KUKA KRL program: Glode_HanGao.src, Glode_HanGao.dat

--- Glode_HanGao.src ---
&ACCESS RVO1
&REL 506
&PARAM EDITMASK = *
&PARAM TEMPLATE = C:\KRC\Roboter\Template\vorgabe
&PARAM DISKPATH = KRC:\R1\Program\HG
DEF Glode_HanGao( )

;# DATE:2021-1-4


END



GLOBAL DEF Vision_Path(PATH_POS:OUT,POS_OFFSET:IN)
DECL E6POS PATH_POS,POS_OFFSET

;Halt


IF Vision_OFFSET_STATE==FALSE THEN
 PATH_POS=POS_OFFSET:PATH_POS
ENDIF

Vision_OFFSET_STATE=TRUE



END
GLOBAL DEF Vision_EndPath(PATH_POS:OUT,POS_OFFSET:IN)
DECL E6POS PATH_POS,POS_OFFSET

;HALT
INTERRUPT OFF 20
PATH_POS=INV_Pos(POS_OFFSET):PATH_POS



END



GLOBAL DEF Vision_Results_Pos(Vision_PATH:IN,Result_Pos:IN,POS_Offset:OUT)
DECL E6POS POS_Offset,Result_Pos,Offset,Error_Offset,Result_Pos_Inv
DECL Vision_PATH_Enum Vision_PATH
DECL INT Result_ID,OPFFSET
DECL CHAR POS_Sting[1024],Message_Show[1024]
DECL State_t _State
DECL VAR_STATE VarT

Message_Show[]=" "
OPFFSET=0
Offset=$NULLFRAME
Error_Offset=$NULLFRAME

IF Vision_Type ==#Vision_Run THEN


VarT=VARSTATE("POS_Offset")
SWITCH VarT

CASE #DECLARED

RETURN

CASE #INITIALIZED

;Result_Pos_Inv=Inv_Pos(Result_Pos)

Error_Offset=Inv_Pos(Result_Pos):Pos_Offset
;Halt

;Offset.X=Error_Offset.X-POS_Offset.X
;Offset.Y=Error_Offset.Y-POS_Offset.Y
;Offset.Z=Error_Offset.z-POS_Offset.Z
;Offset.A=Error_Offset.A-POS_Offset.A
;Offset.B=Error_Offset.B-POS_Offset.B
;Offset.C=Error_Offset.C-POS_Offset.C





SWITCH Vision_PATH
CASE #X

SWRITE( Message_Show[] , _State , OPFFSET ,"Vision Find  Offset: X:%7.3F Translation Max:%7.3F," ,Error_Offset.X, Vision_Trans_Max_Offset  )

if (ABS(Error_Offset.X)<Vision_Trans_Max_Offset)  THEN

POS_Offset.X=Result_Pos.X
ELSE


MsgQuit(Message_Show[], "HanGao")
RETURN
ENDIF


CASE #Y

SWRITE( Message_Show[] , _State , OPFFSET ,"Vision Find  Offset: Y:%7.3F Translation Max:%7.3F," ,Error_Offset.Y, Vision_Trans_Max_Offset  )
if (ABS(Error_Offset.Y)<Vision_Trans_Max_Offset)  THEN

POS_Offset.Y=Result_Pos.Y
ELSE


MsgQuit(Message_Show[], "HanGao")
RETURN
ENDIF
CASE #Z
SWRITE( Message_Show[] , _State , OPFFSET ,"Vision Find  Offset: Z:%7.3F Translation Max:%7.3F," ,Error_Offset.Z, Vision_Trans_Max_Offset  )
if (ABS(Error_Offset.Z)<Vision_Trans_Max_Offset)  THEN

POS_Offset.Z=Result_Pos.Z
ELSE


MsgQuit(Message_Show[], "HanGao")
RETURN
ENDIF
CASE #XY

SWRITE( Message_Show[] , _State , OPFFSET ,"Vision Find  Offset: X:%7.3F,Y:%7.3F Translation Max:%7.3F" ,Error_Offset.X,Error_Offset.Y ,Vision_Trans_Max_Offset  )

if (ABS(Error_Offset.X)<Vision_Trans_Max_Offset) AND (ABS(Error_Offset.Y)<Vision_Trans_Max_Offset)  THEN

POS_Offset.X=Result_Pos.X
POS_Offset.Y=Result_Pos.Y
ELSE


MsgQuit(Message_Show[], "HanGao")
RETURN
ENDIF
CASE #XZ

SWRITE( Message_Show[] , _State , OPFFSET ,"Vision Find  Offset: X:%7.3F,Z:%7.3F Translation Max:%7.3F" ,Error_Offset.X,Error_Offset.Z, Vision_Trans_Max_Offset  )

if (ABS(Error_Offset.X)<Vision_Trans_Max_Offset) AND (ABS(Error_Offset.Z)<Vision_Trans_Max_Offset)  THEN

POS_Offset.X=Result_Pos.X
POS_Offset.Z=Result_Pos.Z
ELSE


MsgQuit(Message_Show[], "HanGao")
RETURN
ENDIF
CASE #YZ

SWRITE( Message_Show[] , _State , OPFFSET ,"Vision Find  Offset: Y:%7.3F,Z:%7.3F Translation Max:%7.3F" ,Error_Offset.Y,Error_Offset.Z, Vision_Trans_Max_Offset  )

if (ABS(Error_Offset.Y)<Vision_Trans_Max_Offset) AND (ABS(Error_Offset.Y)<Vision_Trans_Max_Offset)  THEN

POS_Offset.Y=Result_Pos.Y
POS_Offset.Z=Result_Pos.Z
ELSE


MsgQuit(Message_Show[], "HanGao")
RETURN
ENDIF
CASE #XYZ

SWRITE( Message_Show[] , _State , OPFFSET ,"Vision Find  Offset: X:%7.3F,Y:%7.3F,Z:%7.3F Translation Max:%7.3F" ,Error_Offset.X,Error_Offset.Y,Error_Offset.Z, Vision_Trans_Max_Offset  )

if (ABS(Error_Offset.X)<Vision_Trans_Max_Offset) AND (ABS(Error_Offset.Y)<Vision_Trans_Max_Offset) AND (ABS(Error_Offset.Z)<Vision_Trans_Max_Offset)   THEN

POS_Offset.X=Result_Pos.X
POS_Offset.Y=Result_Pos.Y
POS_Offset.Z=Result_Pos.Z
ELSE


MsgQuit(Message_Show[], "HanGao")
RETURN
ENDIF
CASE #XYZABC

SWRITE( Message_Show[] , _State , OPFFSET ,"Vision Find  Offset: X:%7.3F,Y:%7.3F,Z:%7.3F,A:%7.3F,B:%7.3F,C:%7.3F Translation Max:%7.3F,Rotation Max:%7.3F" ,Error_Offset.X,Error_Offset.Y,Error_Offset.Z,Error_Offset.A,Error_Offset.B,Error_Offset.C, Vision_Trans_Max_Offset ,Vision_Rota_Max_Offset )


if (ABS(Error_Offset.X)<Vision_Trans_Max_Offset) AND (ABS(Error_Offset.Y)<Vision_Trans_Max_Offset) AND (ABS(Error_Offset.Z)<Vision_Trans_Max_Offset) AND (ABS(Error_Offset.A)<Vision_Rota_Max_Offset) AND (ABS(Error_Offset.B)<Vision_Rota_Max_Offset) AND (ABS(Error_Offset.C)<Vision_Rota_Max_Offset)  THEN

POS_Offset.X=Result_Pos.X
POS_Offset.Y=Result_Pos.Y
POS_Offset.Z=Result_Pos.Z
POS_Offset.A=Result_Pos.A
POS_Offset.B=Result_Pos.B
POS_Offset.C=Result_Pos.C

ELSE

MsgQuit(Message_Show[], "HanGao")
RETURN
ENDIF
ENDSWITCH



MSGNOTIFY(Message_Show[])



CASE #UNKNOWN

RETURN

ENDSWITCH


ENDIF



;ENDIF

END
GLOBAL DEF Vision_Results_Offset(Vision_PATH:IN,POS_Offset_1:OUT,POS_Offset_2:OUT,POS_Offset_3:OUT,POS_Offset_4:OUT,POS_Offset_5:OUT,POS_Offset_6:OUT,POS_Offset_7:OUT,POS_Offset_8:OUT,POS_Offset_9:OUT)
DECL E6POS POS_Offset_1 ,POS_Offset_2,POS_Offset_3,POS_Offset_4,POS_Offset_5,POS_Offset_6,POS_Offset_7,POS_Offset_8,POS_Offset_9
DECL Vision_PATH_Enum Vision_PATH
DECL INT Result_ID

IF Vision_Type ==#Vision_Run THEN



Vision_Results_Pos(Vision_PATH,Vision_Result_POS,POS_Offset_1)
Vision_Results_Pos(Vision_PATH,Vision_Result_POS,POS_Offset_2)
Vision_Results_Pos(Vision_PATH,Vision_Result_POS,POS_Offset_3)
Vision_Results_Pos(Vision_PATH,Vision_Result_POS,POS_Offset_4)
Vision_Results_Pos(Vision_PATH,Vision_Result_POS,POS_Offset_5)
Vision_Results_Pos(Vision_PATH,Vision_Result_POS,POS_Offset_6)
Vision_Results_Pos(Vision_PATH,Vision_Result_POS,POS_Offset_7)
Vision_Results_Pos(Vision_PATH,Vision_Result_POS,POS_Offset_8)
Vision_Results_Pos(Vision_PATH,Vision_Result_POS,POS_Offset_9)
ENDIF




END






GLOBAL DEF HanGao_Surr_Calculate(Surr_Path:IN , Sink_Area:IN ,POS_Type:IN , Lin_Pos:OUt , Cir_Middle_POS:OUT , Cir_END_POS:OUT , Offset_info:OUT  ,Offset_cir_info:out , Offset_No:IN , Work_Area:IN, Sink_Type:IN)
;------------DECL_VALUE--------------
DECL REAL Surr_Path
DECL Sink_Type_Enum  Sink_Type
DECL Area_Enum Sink_Area
DECL E6POS Lin_Pos
DECL E6POS Cir_Middle_POS
DECL E6POS Cir_END_POS
DECL Pos_Type_Enum Pos_Type
DECL Offset_POS Offset_info , Offset_cir_info
DECL Surround_Welding_Type Sink_Welding_Size
DECL INT OFFSET_NO,Work_Area

;------------DECL_VALUE--------------





Lin_Pos={X 0,Y 0, Z 0,A 0,B 0,C 0}

Cir_Middle_POS={X 0,Y 0, Z 0,A 0,B 0,C 0}

Cir_END_POS={X 0,Y 0, Z 0,A 0,B 0,C 0}


switch Work_Area

CASE 1
Sink_Welding_Size=N1_Sink_Data

CASE 2
Sink_Welding_Size=N2_Sink_Data

ENDSWITCH



SWITCH Sink_Area

CASE #L0





 UL_Equation(N315_OFFSET_POS,N45_OFFSET_POS,(Surr_Path*0.01),Sink_Welding_Size.Sink_Size_R,Lin_Pos)



 ;Lin_Pos.X=Sink_Welding_Size.Sink_Size_Width+Sink_Welding_Size.Sink_Size_Down_Distance
 ;Lin_Pos.Y=(Sink_Welding_Size.Sink_Size_Long-Sink_Welding_Size.Sink_Size_R*2)* (1-(Surr_Path*0.01))+Sink_Welding_Size.Sink_Size_Left_Distance+Sink_Welding_Size.Sink_Size_R
 Lin_Pos.Z=-(Sink_Welding_Size.Sink_Size_Panel_Thick)

 Lin_Pos.A=0
 Lin_Pos.B=L0_Welding_Craft[Work_Area,OFFSET_NO].Welding_Angle
 Lin_Pos.C=0


L0_Welding_Craft[Work_Area,OFFSET_NO].Welding_Pos.X=Lin_Pos.X
L0_Welding_Craft[Work_Area,OFFSET_NO].Welding_Pos.Y=Lin_Pos.Y
L0_Welding_Craft[Work_Area,OFFSET_NO].Welding_Pos.Z=Lin_Pos.Z
L0_Welding_Craft[Work_Area,OFFSET_NO].Welding_Pos.A=Lin_Pos.A
L0_Welding_Craft[Work_Area,OFFSET_NO].Welding_Pos.B=Lin_Pos.B
L0_Welding_Craft[Work_Area,OFFSET_NO].Welding_Pos.C=Lin_Pos.C
CASE #C45


SWITCH Pos_Type

CASE #C_LIN_POS


UL_Equation(N315_OFFSET_POS,N45_OFFSET_POS,1,Sink_Welding_Size.Sink_Size_R,Lin_Pos)

;Lin_Pos.X=Sink_Welding_Size.Sink_Size_Width+Sink_Welding_Size.Sink_Size_Down_Distance
;Lin_Pos.Y=Sink_Welding_Size.Sink_Size_Left_Distance+Sink_Welding_Size.Sink_Size_R
Lin_Pos.Z=-(Sink_Welding_Size.Sink_Size_Panel_Thick)

Lin_Pos.A=0
Lin_Pos.B=C45_Welding_Craft[Work_Area,1].Welding_Angle
Lin_Pos.C=0

C45_Welding_Craft[Work_Area,1].Welding_Pos.X=Lin_Pos.X
C45_Welding_Craft[Work_Area,1].Welding_Pos.Y=Lin_Pos.Y
C45_Welding_Craft[Work_Area,1].Welding_Pos.Z=Lin_Pos.Z
C45_Welding_Craft[Work_Area,1].Welding_Pos.A=Lin_Pos.A
C45_Welding_Craft[Work_Area,1].Welding_Pos.B=Lin_Pos.B
C45_Welding_Craft[Work_Area,1].Welding_Pos.C=Lin_Pos.C

CASE #C_CIR_POS


 Cir_Middle_POS.X=N45_CIR_POS.x
 Cir_Middle_POS.Y=N45_CIR_POS.Y

 ;Cir_Middle_POS.x=Sink_Welding_Size.Sink_Size_Down_Distance+Sink_Welding_Size.Sink_Size_Width-Sink_Welding_Size.Sink_Size_R+(COS(45)*Sink_Welding_Size.Sink_Size_R)
 ;Cir_Middle_POS.Y=Sink_Welding_Size.Sink_Size_Left_Distance+((1-COS(45))*Sink_Welding_Size.Sink_Size_R)
 Cir_Middle_POS.Z=-(Sink_Welding_Size.Sink_Size_Panel_Thick)


 UL_Equation(N45_OFFSET_POS,N135_OFFSET_POS,0,Sink_Welding_Size.Sink_Size_R,Cir_END_POS)

 ;Cir_END_POS.X=Sink_Welding_Size.Sink_Size_Down_Distance+Sink_Welding_Size.Sink_Size_Width-Sink_Welding_Size.Sink_Size_R
 ;Cir_END_POS.Y=Sink_Welding_Size.Sink_Size_Left_Distance
 Cir_END_POS.Z=-(Sink_Welding_Size.Sink_Size_Panel_Thick)


 Cir_END_POS.A=0
 Cir_END_POS.B=0
 Cir_END_POS.C=C45_Welding_Craft[Work_Area,3].Welding_Angle



C45_Welding_Craft[Work_Area,2].Welding_Pos.X=Cir_Middle_POS.X
C45_Welding_Craft[Work_Area,2].Welding_Pos.Y=Cir_Middle_POS.Y
C45_Welding_Craft[Work_Area,2].Welding_Pos.Z=Cir_Middle_POS.Z
C45_Welding_Craft[Work_Area,2].Welding_Pos.A=Cir_Middle_POS.A
C45_Welding_Craft[Work_Area,2].Welding_Pos.B=Cir_Middle_POS.B
C45_Welding_Craft[Work_Area,2].Welding_Pos.C=Cir_Middle_POS.C

C45_Welding_Craft[Work_Area,3].Welding_Pos.X=Cir_END_POS.X
C45_Welding_Craft[Work_Area,3].Welding_Pos.Y=Cir_END_POS.Y
C45_Welding_Craft[Work_Area,3].Welding_Pos.Z=Cir_END_POS.Z
C45_Welding_Craft[Work_Area,3].Welding_Pos.A=Cir_END_POS.A
C45_Welding_Craft[Work_Area,3].Welding_Pos.B=Cir_END_POS.B
C45_Welding_Craft[Work_Area,3].Welding_Pos.C=Cir_END_POS.C

ENDSWITCH


CASE #L90


UL_Equation(N45_OFFSET_POS,N135_OFFSET_POS,(Surr_Path*0.01),Sink_Welding_Size.Sink_Size_R, Lin_Pos)

 ;Lin_Pos.X=(Sink_Welding_Size.Sink_Size_Width-Sink_Welding_Size.Sink_Size_R*2)* (1-(Surr_Path*0.01))+Sink_Welding_Size.Sink_Size_Down_Distance+Sink_Welding_Size.Sink_Size_R
 ;Lin_Pos.Y=Sink_Welding_Size.Sink_Size_Left_Distance
 Lin_Pos.Z=-(Sink_Welding_Size.Sink_Size_Panel_Thick)
 Lin_Pos.A=0
 Lin_Pos.B=0
 Lin_Pos.C=L90_Welding_Craft[Work_Area,OFFSET_NO].Welding_Angle

L90_Welding_Craft[Work_Area,OFFSET_NO].Welding_Pos.X=Lin_Pos.X
L90_Welding_Craft[Work_Area,OFFSET_NO].Welding_Pos.Y=Lin_Pos.Y
L90_Welding_Craft[Work_Area,OFFSET_NO].Welding_Pos.Z=Lin_Pos.Z
L90_Welding_Craft[Work_Area,OFFSET_NO].Welding_Pos.A=Lin_Pos.A
L90_Welding_Craft[Work_Area,OFFSET_NO].Welding_Pos.B=Lin_Pos.B
L90_Welding_Craft[Work_Area,OFFSET_NO].Welding_Pos.C=Lin_Pos.C

CASE #C135

SWITCH Pos_Type

CASE #C_LIN_POS

UL_Equation(N45_OFFSET_POS,N135_OFFSET_POS,1,Sink_Welding_Size.Sink_Size_R, Lin_Pos)

 ;Lin_Pos.X=Sink_Welding_Size.Sink_Size_Down_Distance+Sink_Welding_Size.Sink_Size_R
 ;Lin_Pos.Y=Sink_Welding_Size.Sink_Size_Left_Distance
 Lin_Pos.Z=-(Sink_Welding_Size.Sink_Size_Panel_Thick)
 Lin_Pos.A=0
 Lin_Pos.B=0
 Lin_Pos.C=C135_Welding_Craft[Work_Area,1].Welding_Angle

C135_Welding_Craft[Work_Area,1].Welding_Pos.X=Lin_Pos.X
C135_Welding_Craft[Work_Area,1].Welding_Pos.Y=Lin_Pos.Y
C135_Welding_Craft[Work_Area,1].Welding_Pos.Z=Lin_Pos.Z
C135_Welding_Craft[Work_Area,1].Welding_Pos.A=Lin_Pos.A
C135_Welding_Craft[Work_Area,1].Welding_Pos.B=Lin_Pos.B
C135_Welding_Craft[Work_Area,1].Welding_Pos.C=Lin_Pos.C

CASE #C_CIR_POS



 Cir_Middle_POS.X=N135_CIR_POS.x
 Cir_Middle_POS.Y=N135_CIR_POS.Y


 ;Cir_Middle_POS.x=Sink_Welding_Size.Sink_Size_Down_Distance+((1-COS(45))*Sink_Welding_Size.Sink_Size_R)
 ;Cir_Middle_POS.Y=Sink_Welding_Size.Sink_Size_Left_Distance+((1-COS(45))*Sink_Welding_Size.Sink_Size_R)
 Cir_Middle_POS.Z=-(Sink_Welding_Size.Sink_Size_Panel_Thick)



 UL_Equation(N135_OFFSET_POS,N225_OFFSET_POS,0,Sink_Welding_Size.Sink_Size_R,Cir_END_POS)

 ;Cir_END_POS.X=Sink_Welding_Size.Sink_Size_Down_Distance
 ;Cir_END_POS.Y=Sink_Welding_Size.Sink_Size_Left_Distance+Sink_Welding_Size.Sink_Size_R
 Cir_END_POS.Z=-(Sink_Welding_Size.Sink_Size_Panel_Thick)
 Cir_END_POS.A=0
 Cir_END_POS.B=C135_Welding_Craft[Work_Area,3].Welding_Angle
 Cir_END_POS.C=0

C135_Welding_Craft[Work_Area,2].Welding_Pos.X=Cir_Middle_POS.X
C135_Welding_Craft[Work_Area,2].Welding_Pos.Y=Cir_Middle_POS.Y
C135_Welding_Craft[Work_Area,2].Welding_Pos.Z=Cir_Middle_POS.Z
C135_Welding_Craft[Work_Area,2].Welding_Pos.A=Cir_Middle_POS.A
C135_Welding_Craft[Work_Area,2].Welding_Pos.B=Cir_Middle_POS.B
C135_Welding_Craft[Work_Area,2].Welding_Pos.C=Cir_Middle_POS.C

C135_Welding_Craft[Work_Area,3].Welding_Pos.X=Cir_END_POS.X
C135_Welding_Craft[Work_Area,3].Welding_Pos.Y=Cir_END_POS.Y
C135_Welding_Craft[Work_Area,3].Welding_Pos.Z=Cir_END_POS.Z
C135_Welding_Craft[Work_Area,3].Welding_Pos.A=Cir_END_POS.A
C135_Welding_Craft[Work_Area,3].Welding_Pos.B=Cir_END_POS.B
C135_Welding_Craft[Work_Area,3].Welding_Pos.C=Cir_END_POS.C

ENDSWITCH


CASE #L180

UL_Equation(N135_OFFSET_POS,N225_OFFSET_POS,(Surr_Path*0.01),Sink_Welding_Size.Sink_Size_R, Lin_Pos)

 ;Lin_Pos.X=Sink_Welding_Size.Sink_Size_Down_Distance
 ;Lin_Pos.Y=(Sink_Welding_Size.Sink_Size_Long-Sink_Welding_Size.Sink_Size_R*2)* (Surr_Path*0.01)+Sink_Welding_Size.Sink_Size_Left_Distance+Sink_Welding_Size.Sink_Size_R
 Lin_Pos.Z=-(Sink_Welding_Size.Sink_Size_Panel_Thick)
 Lin_Pos.A=0
 Lin_Pos.B=L180_Welding_Craft[Work_Area,OFFSET_NO].Welding_Angle
 Lin_Pos.C=0

L180_Welding_Craft[Work_Area,OFFSET_NO].Welding_Pos.X=Lin_Pos.X
L180_Welding_Craft[Work_Area,OFFSET_NO].Welding_Pos.Y=Lin_Pos.Y
L180_Welding_Craft[Work_Area,OFFSET_NO].Welding_Pos.Z=Lin_Pos.Z
L180_Welding_Craft[Work_Area,OFFSET_NO].Welding_Pos.A=Lin_Pos.A
L180_Welding_Craft[Work_Area,OFFSET_NO].Welding_Pos.B=Lin_Pos.B
L180_Welding_Craft[Work_Area,OFFSET_NO].Welding_Pos.C=Lin_Pos.C

CASE #C225

SWITCH Pos_Type

CASE #C_LIN_POS


 UL_Equation(N135_OFFSET_POS,N225_OFFSET_POS,1,Sink_Welding_Size.Sink_Size_R, Lin_Pos)

 ;Lin_Pos.X=Sink_Welding_Size.Sink_Size_Down_Distance
 ;Lin_Pos.Y=Sink_Welding_Size.Sink_Size_Left_Distance+Sink_Welding_Size.Sink_Size_Long-Sink_Welding_Size.Sink_Size_R
 Lin_Pos.Z=-(Sink_Welding_Size.Sink_Size_Panel_Thick)
 Lin_Pos.A=0
 Lin_Pos.B=C225_Welding_Craft[Work_Area,1].Welding_Angle
 Lin_Pos.C=0

C225_Welding_Craft[Work_Area,1].Welding_Pos.X=Lin_Pos.X
C225_Welding_Craft[Work_Area,1].Welding_Pos.Y=Lin_Pos.Y
C225_Welding_Craft[Work_Area,1].Welding_Pos.Z=Lin_Pos.Z
C225_Welding_Craft[Work_Area,1].Welding_Pos.A=Lin_Pos.A
C225_Welding_Craft[Work_Area,1].Welding_Pos.B=Lin_Pos.B
C225_Welding_Craft[Work_Area,1].Welding_Pos.C=Lin_Pos.C

CASE #C_CIR_POS


 Cir_Middle_POS.X=N225_CIR_POS.x
 Cir_Middle_POS.Y=N225_CIR_POS.Y




 ;Cir_Middle_POS.x=Sink_Welding_Size.Sink_Size_Down_Distance+((1-COS(45))*Sink_Welding_Size.Sink_Size_R)
 ;Cir_Middle_POS.Y=Sink_Welding_Size.Sink_Size_Left_Distance+Sink_Welding_Size.Sink_Size_Long-Sink_Welding_Size.Sink_Size_R+( COS(45)*Sink_Welding_Size.Sink_Size_R )
 Cir_Middle_POS.Z=-(Sink_Welding_Size.Sink_Size_Panel_Thick)

  UL_Equation(N225_OFFSET_POS,N315_OFFSET_POS,0,Sink_Welding_Size.Sink_Size_R,Cir_END_POS)

 ;Cir_END_POS.X=Sink_Welding_Size.Sink_Size_Down_Distance+Sink_Welding_Size.Sink_Size_R
; Cir_END_POS.Y=Sink_Welding_Size.Sink_Size_Left_Distance+Sink_Welding_Size.Sink_Size_Long
 Cir_END_POS.Z=-(Sink_Welding_Size.Sink_Size_Panel_Thick)
 Cir_END_POS.A=0
 Cir_END_POS.B=0
 Cir_END_POS.C=C225_Welding_Craft[Work_Area,3].Welding_Angle

C225_Welding_Craft[Work_Area,2].Welding_Pos.X=Cir_Middle_POS.X
C225_Welding_Craft[Work_Area,2].Welding_Pos.Y=Cir_Middle_POS.Y
C225_Welding_Craft[Work_Area,2].Welding_Pos.Z=Cir_Middle_POS.Z
C225_Welding_Craft[Work_Area,2].Welding_Pos.A=Cir_Middle_POS.A
C225_Welding_Craft[Work_Area,2].Welding_Pos.B=Cir_Middle_POS.B
C225_Welding_Craft[Work_Area,2].Welding_Pos.C=Cir_Middle_POS.C

C225_Welding_Craft[Work_Area,3].Welding_Pos.X=Cir_END_POS.X
C225_Welding_Craft[Work_Area,3].Welding_Pos.Y=Cir_END_POS.Y
C225_Welding_Craft[Work_Area,3].Welding_Pos.Z=Cir_END_POS.Z
C225_Welding_Craft[Work_Area,3].Welding_Pos.A=Cir_END_POS.A
C225_Welding_Craft[Work_Area,3].Welding_Pos.B=Cir_END_POS.B
C225_Welding_Craft[Work_Area,3].Welding_Pos.C=Cir_END_POS.C

ENDSWITCH


CASE #L270



UL_Equation(N225_OFFSET_POS,N315_OFFSET_POS,(Surr_Path*0.01),Sink_Welding_Size.Sink_Size_R, Lin_Pos)




; Lin_Pos.X=(Sink_Welding_Size.Sink_Size_Width-Sink_Welding_Size.Sink_Size_R*2)* (Surr_Path*0.01)+Sink_Welding_Size.Sink_Size_Down_Distance+Sink_Welding_Size.Sink_Size_R
 ;Lin_Pos.Y=Sink_Welding_Size.Sink_Size_Left_Distance+Sink_Welding_Size.Sink_Size_Long
 Lin_Pos.Z=-(Sink_Welding_Size.Sink_Size_Panel_Thick)
 Lin_Pos.A=0
 Lin_Pos.B=0
 Lin_Pos.C=L270_Welding_Craft[Work_Area,OFFSET_NO].Welding_Angle

L270_Welding_Craft[Work_Area,OFFSET_NO].Welding_Pos.X=Lin_Pos.X
L270_Welding_Craft[Work_Area,OFFSET_NO].Welding_Pos.Y=Lin_Pos.Y
L270_Welding_Craft[Work_Area,OFFSET_NO].Welding_Pos.Z=Lin_Pos.Z
L270_Welding_Craft[Work_Area,OFFSET_NO].Welding_Pos.A=Lin_Pos.A
L270_Welding_Craft[Work_Area,OFFSET_NO].Welding_Pos.B=Lin_Pos.B
L270_Welding_Craft[Work_Area,OFFSET_NO].Welding_Pos.C=Lin_Pos.C

CASE #C315

SWITCH Pos_Type

CASE #C_LIN_POS



 UL_Equation(N225_OFFSET_POS,N315_OFFSET_POS,1,Sink_Welding_Size.Sink_Size_R, Lin_Pos)




 ;Lin_Pos.X=Sink_Welding_Size.Sink_Size_Down_Distance+Sink_Welding_Size.Sink_Size_Width-Sink_Welding_Size.Sink_Size_R
 ;Lin_Pos.Y=Sink_Welding_Size.Sink_Size_Long+Sink_Welding_Size.Sink_Size_Left_Distance
 Lin_Pos.Z=-(Sink_Welding_Size.Sink_Size_Panel_Thick)
 Lin_Pos.A=0
 Lin_Pos.B=0
 Lin_Pos.C=C315_Welding_Craft[Work_Area,1].Welding_Angle

 C315_Welding_Craft[Work_Area,1].Welding_Pos.X=Lin_Pos.X
 C315_Welding_Craft[Work_Area,1].Welding_Pos.Y=Lin_Pos.Y
 C315_Welding_Craft[Work_Area,1].Welding_Pos.Z=Lin_Pos.Z
 C315_Welding_Craft[Work_Area,1].Welding_Pos.A=Lin_Pos.A
 C315_Welding_Craft[Work_Area,1].Welding_Pos.B=Lin_Pos.B
 C315_Welding_Craft[Work_Area,1].Welding_Pos.C=Lin_Pos.C

CASE #C_CIR_POS


 Cir_Middle_POS.X=N315_CIR_POS.x
 Cir_Middle_POS.Y=N315_CIR_POS.Y


 ;Cir_Middle_POS.x=Sink_Welding_Size.Sink_Size_Down_Distance+Sink_Welding_Size.Sink_Size_Width-Sink_Welding_Size.Sink_Size_R+(COS(45)*Sink_Welding_Size.Sink_Size_R)
 ;Cir_Middle_POS.Y=Sink_Welding_Size.Sink_Size_Long+Sink_Welding_Size.Sink_Size_Left_Distance-Sink_Welding_Size.Sink_Size_R+(COS(45)*Sink_Welding_Size.Sink_Size_R)
 Cir_Middle_POS.Z=-(Sink_Welding_Size.Sink_Size_Panel_Thick)

   UL_Equation(N315_OFFSET_POS,N45_OFFSET_POS,0,Sink_Welding_Size.Sink_Size_R,Cir_END_POS)

 ;Cir_END_POS.X=Sink_Welding_Size.Sink_Size_Down_Distance+Sink_Welding_Size.Sink_Size_Width
 ;Cir_END_POS.Y=Sink_Welding_Size.Sink_Size_Left_Distance+Sink_Welding_Size.Sink_Size_Long-Sink_Welding_Size.Sink_Size_R
 Cir_END_POS.Z=-(Sink_Welding_Size.Sink_Size_Panel_Thick)
 Cir_END_POS.A=0
 Cir_END_POS.B=C315_Welding_Craft[Work_Area,3].Welding_Angle
 Cir_END_POS.C=0

C315_Welding_Craft[Work_Area,2].Welding_Pos.X=Cir_Middle_POS.X
C315_Welding_Craft[Work_Area,2].Welding_Pos.Y=Cir_Middle_POS.Y
C315_Welding_Craft[Work_Area,2].Welding_Pos.Z=Cir_Middle_POS.Z
C315_Welding_Craft[Work_Area,2].Welding_Pos.A=Cir_Middle_POS.A
C315_Welding_Craft[Work_Area,2].Welding_Pos.B=Cir_Middle_POS.B
C315_Welding_Craft[Work_Area,2].Welding_Pos.C=Cir_Middle_POS.C

C315_Welding_Craft[Work_Area,3].Welding_Pos.X=Cir_END_POS.X
C315_Welding_Craft[Work_Area,3].Welding_Pos.Y=Cir_END_POS.Y
C315_Welding_Craft[Work_Area,3].Welding_Pos.Z=Cir_END_POS.Z
C315_Welding_Craft[Work_Area,3].Welding_Pos.A=Cir_END_POS.A
C315_Welding_Craft[Work_Area,3].Welding_Pos.B=Cir_END_POS.B
C315_Welding_Craft[Work_Area,3].Welding_Pos.C=Cir_END_POS.C

ENDSWITCH





CASE #N45
;




SWITCH  Offset_No

CASE 1

SWITCH Sink_Welding_Size.Sink_Type
CASE #UpDown_One

Lin_Pos.X=D45_Start_POS.X
Lin_Pos.Y=D45_Start_POS.X

;Lin_Pos.X=Sink_Welding_Size.Sink_Size_Down_Distance*2+Sink_Welding_Size.Sink_Size_Width
;Lin_Pos.Y=Sink_Welding_Size.Sink_Size_Short_TwoPos
Lin_Pos.Z=-150.000
Lin_Pos.A=0
Lin_Pos.B=0
Lin_Pos.C=0
case #LeftRight_One

Lin_Pos.X=D45_Start_POS.X
Lin_Pos.Y=D45_Start_POS.Y

;Lin_Pos.X=Sink_Welding_Size.Sink_Size_Short_OnePos+Sink_Welding_Size.Sink_Size_Short_TwoPos
;Lin_Pos.Y=0
Lin_Pos.Z=-150.000
Lin_Pos.A=0
Lin_Pos.B=0
Lin_Pos.C=0
ENDSWITCH

N45_Short_Craft[Work_Area,1].Welding_Pos.X=Lin_Pos.X
N45_Short_Craft[Work_Area,1].Welding_Pos.Y=Lin_Pos.Y
N45_Short_Craft[Work_Area,1].Welding_Pos.Z=Lin_Pos.Z
N45_Short_Craft[Work_Area,1].Welding_Pos.A=Lin_Pos.A
N45_Short_Craft[Work_Area,1].Welding_Pos.B=Lin_Pos.B
N45_Short_Craft[Work_Area,1].Welding_Pos.C=Lin_Pos.C

CASE 2
SWITCH Sink_Welding_Size.Sink_Type
CASE #UpDown_One

Lin_Pos.X=D45_Start_POS.X
Lin_Pos.Y=D45_Start_POS.Y

;Lin_Pos.X=Sink_Welding_Size.Sink_Size_Down_Distance*2+Sink_Welding_Size.Sink_Size_Width
;Lin_Pos.Y=Sink_Welding_Size.Sink_Size_Short_TwoPos
Lin_Pos.Z=0
Lin_Pos.A=0
Lin_Pos.B=0
Lin_Pos.C=0
case #LeftRight_One

Lin_Pos.X=D45_Start_POS.X
Lin_Pos.Y=D45_Start_POS.Y

; Lin_Pos.X=Sink_Welding_Size.Sink_Size_Short_OnePos+Sink_Welding_Size.Sink_Size_Short_TwoPos
; Lin_Pos.Y=0
Lin_Pos.Z=0
Lin_Pos.A=0
Lin_Pos.B=0
Lin_Pos.C=0
ENDSWITCH


N45_Short_Craft[Work_Area,2].Welding_Pos.X=Lin_Pos.X
N45_Short_Craft[Work_Area,2].Welding_Pos.Y=Lin_Pos.Y
N45_Short_Craft[Work_Area,2].Welding_Pos.Z=Lin_Pos.Z
N45_Short_Craft[Work_Area,2].Welding_Pos.A=Lin_Pos.A
N45_Short_Craft[Work_Area,2].Welding_Pos.B=Lin_Pos.B
N45_Short_Craft[Work_Area,2].Welding_Pos.C=Lin_Pos.C

CASE 3
SWITCH Sink_Welding_Size.Sink_Type
CASE #UpDown_One

Lin_Pos.X=D45_End_POS.X
Lin_Pos.Y=D45_End_POS.Y

;Lin_Pos.X=Sink_Welding_Size.Sink_Size_Down_Distance*2+Sink_Welding_Size.Sink_Size_Width
;Lin_Pos.Y=Sink_Welding_Size.Sink_Size_Short_TwoPos-Sink_Welding_Size.Sink_Size_Short_Side
Lin_Pos.Z=0.000
Lin_Pos.A=0
Lin_Pos.B=0
Lin_Pos.C=0
case #LeftRight_One

Lin_Pos.X=D45_End_POS.X
Lin_Pos.Y=D45_End_POS.Y

;Lin_Pos.X=Sink_Welding_Size.Sink_Size_Short_OnePos+Sink_Welding_Size.Sink_Size_Short_TwoPos
;Lin_Pos.Y=Sink_Welding_Size.Sink_Size_Short_Side
Lin_Pos.Z=0.000
Lin_Pos.A=0
Lin_Pos.B=0
Lin_Pos.C=0
ENDSWITCH


N45_Short_Craft[Work_Area,3].Welding_Pos.X=Lin_Pos.X
N45_Short_Craft[Work_Area,3].Welding_Pos.Y=Lin_Pos.Y
N45_Short_Craft[Work_Area,3].Welding_Pos.Z=Lin_Pos.Z
N45_Short_Craft[Work_Area,3].Welding_Pos.A=Lin_Pos.A
N45_Short_Craft[Work_Area,3].Welding_Pos.B=Lin_Pos.B
N45_Short_Craft[Work_Area,3].Welding_Pos.C=Lin_Pos.C

CASE 4
SWITCH Sink_Welding_Size.Sink_Type
CASE #UpDown_One

UL_Equation(D45_Start_POS,D45_End_POS,(Surr_Path*0.01),Sink_Welding_Size.Sink_Size_R,Lin_Pos)

;Lin_Pos.X=Sink_Welding_Size.Sink_Size_Down_Distance+Sink_Welding_Size.Sink_Size_Width+Sink_Welding_Size.Sink_Size_Short_Side*(Surr_Path/100)
;Lin_Pos.Y=Sink_Welding_Size.Sink_Size_Short_TwoPos-Sink_Welding_Size.Sink_Size_Short_Side
Lin_Pos.Z=-150
Lin_Pos.A=0
Lin_Pos.B=0
Lin_Pos.C=0
case #LeftRight_One

UL_Equation(D45_Start_POS,D45_End_POS,(Surr_Path*0.01),Sink_Welding_Size.Sink_Size_R,Lin_Pos)

;Lin_Pos.X=Sink_Welding_Size.Sink_Size_Short_OnePos+Sink_Welding_Size.Sink_Size_Short_TwoPos
;Lin_Pos.Y=Sink_Welding_Size.Sink_Size_Short_Side-Sink_Welding_Size.Sink_Size_Short_Side*(Surr_Path/100)
Lin_Pos.Z=-150
Lin_Pos.A=0
Lin_Pos.B=0
Lin_Pos.C=0
ENDSWITCH


N45_Short_Craft[Work_Area,4].Welding_Pos.X=Lin_Pos.X
N45_Short_Craft[Work_Area,4].Welding_Pos.Y=Lin_Pos.Y
N45_Short_Craft[Work_Area,4].Welding_Pos.Z=Lin_Pos.Z
N45_Short_Craft[Work_Area,4].Welding_Pos.A=Lin_Pos.A
N45_Short_Craft[Work_Area,4].Welding_Pos.B=Lin_Pos.B
N45_Short_Craft[Work_Area,4].Welding_Pos.C=Lin_Pos.C
ENDSWITCH






CASE #N135
;
SWITCH  Offset_No

CASE 1
SWITCH Sink_Welding_Size.Sink_Type
CASE #UpDown_One

Lin_Pos.X=D135_Start_POS.X
Lin_Pos.Y=D135_Start_POS.Y

;Lin_Pos.X=0
;Lin_Pos.Y=Sink_Welding_Size.Sink_Size_Short_OnePos
Lin_Pos.Z=-150.000
Lin_Pos.A=0
Lin_Pos.B=0
Lin_Pos.C=0
case #LeftRight_One

Lin_Pos.X=D135_Start_POS.X
Lin_Pos.Y=D135_Start_POS.Y

;Lin_Pos.X=Sink_Welding_Size.Sink_Size_Short_OnePos
;Lin_Pos.Y=0
Lin_Pos.Z=-150.000
Lin_Pos.A=0
Lin_Pos.B=0
Lin_Pos.C=0
ENDSWITCH


N135_Short_Craft[Work_Area,1].Welding_Pos.X=Lin_Pos.X
N135_Short_Craft[Work_Area,1].Welding_Pos.Y=Lin_Pos.Y
N135_Short_Craft[Work_Area,1].Welding_Pos.Z=Lin_Pos.Z
N135_Short_Craft[Work_Area,1].Welding_Pos.A=Lin_Pos.A
N135_Short_Craft[Work_Area,1].Welding_Pos.B=Lin_Pos.B
N135_Short_Craft[Work_Area,1].Welding_Pos.C=Lin_Pos.C

CASE 2
SWITCH Sink_Welding_Size.Sink_Type
CASE #UpDown_One

Lin_Pos.X=D135_Start_POS.X
Lin_Pos.Y=D135_Start_POS.Y

;Lin_Pos.X=0
;Lin_Pos.Y=Sink_Welding_Size.Sink_Size_Short_OnePos
Lin_Pos.Z=0
Lin_Pos.A=0
Lin_Pos.B=0
Lin_Pos.C=0
case #LeftRight_One

Lin_Pos.X=D135_Start_POS.X
Lin_Pos.Y=D135_Start_POS.Y

;Lin_Pos.X=Sink_Welding_Size.Sink_Size_Short_OnePos
;Lin_Pos.Y=0
Lin_Pos.Z=0
Lin_Pos.A=0
Lin_Pos.B=0
Lin_Pos.C=0
ENDSWITCH


N135_Short_Craft[Work_Area,2].Welding_Pos.X=Lin_Pos.X
N135_Short_Craft[Work_Area,2].Welding_Pos.Y=Lin_Pos.Y
N135_Short_Craft[Work_Area,2].Welding_Pos.Z=Lin_Pos.Z
N135_Short_Craft[Work_Area,2].Welding_Pos.A=Lin_Pos.A
N135_Short_Craft[Work_Area,2].Welding_Pos.B=Lin_Pos.B
N135_Short_Craft[Work_Area,2].Welding_Pos.C=Lin_Pos.C
CASE 3
SWITCH Sink_Welding_Size.Sink_Type
CASE #UpDown_One

Lin_Pos.X=D135_End_POS.X
Lin_Pos.Y=D135_End_POS.Y

;Lin_Pos.X=Sink_Welding_Size.Sink_Size_Short_Side
;Lin_Pos.Y=Sink_Welding_Size.Sink_Size_Short_OnePos
Lin_Pos.Z=0.000
Lin_Pos.A=0
Lin_Pos.B=0
Lin_Pos.C=0
case #LeftRight_One

Lin_Pos.X=D135_End_POS.X
Lin_Pos.Y=D135_End_POS.Y

;Lin_Pos.X=Sink_Welding_Size.Sink_Size_Short_OnePos
;Lin_Pos.Y=Sink_Welding_Size.Sink_Size_Short_Side
Lin_Pos.Z=0.000
Lin_Pos.A=0
Lin_Pos.B=0
Lin_Pos.C=0
ENDSWITCH


N135_Short_Craft[Work_Area,3].Welding_Pos.X=Lin_Pos.X
N135_Short_Craft[Work_Area,3].Welding_Pos.Y=Lin_Pos.Y
N135_Short_Craft[Work_Area,3].Welding_Pos.Z=Lin_Pos.Z
N135_Short_Craft[Work_Area,3].Welding_Pos.A=Lin_Pos.A
N135_Short_Craft[Work_Area,3].Welding_Pos.B=Lin_Pos.B
N135_Short_Craft[Work_Area,3].Welding_Pos.C=Lin_Pos.C
CASE 4
SWITCH Sink_Welding_Size.Sink_Type
CASE #UpDown_One


UL_Equation(D135_Start_POS,D135_End_POS,(Surr_Path*0.01),Sink_Welding_Size.Sink_Size_R,Lin_Pos)

;Lin_Pos.X=Sink_Welding_Size.Sink_Size_Short_Side-Sink_Welding_Size.Sink_Size_Short_Side*(Surr_Path/100)
;Lin_Pos.Y=Sink_Welding_Size.Sink_Size_Short_OnePos
Lin_Pos.Z=-150.000
Lin_Pos.A=0
Lin_Pos.B=0
Lin_Pos.C=0
case #LeftRight_One

UL_Equation(D135_Start_POS,D135_End_POS,(Surr_Path*0.01),Sink_Welding_Size.Sink_Size_R,Lin_Pos)

;Lin_Pos.X=Sink_Welding_Size.Sink_Size_Short_OnePos
;Lin_Pos.Y=Sink_Welding_Size.Sink_Size_Short_Side-Sink_Welding_Size.Sink_Size_Short_Side*(Surr_Path/100)
Lin_Pos.Z=-150.000
Lin_Pos.A=0
Lin_Pos.B=0
Lin_Pos.C=0
ENDSWITCH


N135_Short_Craft[Work_Area,4].Welding_Pos.X=Lin_Pos.X
N135_Short_Craft[Work_Area,4].Welding_Pos.Y=Lin_Pos.Y
N135_Short_Craft[Work_Area,4].Welding_Pos.Z=Lin_Pos.Z
N135_Short_Craft[Work_Area,4].Welding_Pos.A=Lin_Pos.A
N135_Short_Craft[Work_Area,4].Welding_Pos.B=Lin_Pos.B
N135_Short_Craft[Work_Area,4].Welding_Pos.C=Lin_Pos.C

ENDSWITCH





CASE #N225
;
SWITCH  Offset_No

CASE 1
SWITCH Sink_Welding_Size.Sink_Type
CASE #UpDown_One

Lin_Pos.X=D225_Start_POS.X
Lin_Pos.Y=D225_Start_POS.Y

;Lin_Pos.X=0
;Lin_Pos.Y=Sink_Welding_Size.Sink_Size_Short_OnePos+Sink_Welding_Size.Sink_Size_Short_TwoPos
Lin_Pos.Z=-150.000
Lin_Pos.A=0
Lin_Pos.B=0
Lin_Pos.C=0
case #LeftRight_One

Lin_Pos.X=D225_Start_POS.X
Lin_Pos.Y=D225_Start_POS.Y

;Lin_Pos.X=Sink_Welding_Size.Sink_Size_Short_OnePos
;Lin_Pos.Y=Sink_Welding_Size.Sink_Size_Long+Sink_Welding_Size.Sink_Size_Left_Distance*2
Lin_Pos.Z=-150.000
Lin_Pos.A=0
Lin_Pos.B=0
Lin_Pos.C=0
ENDSWITCH


N225_Short_Craft[Work_Area,1].Welding_Pos.X=Lin_Pos.X
N225_Short_Craft[Work_Area,1].Welding_Pos.Y=Lin_Pos.Y
N225_Short_Craft[Work_Area,1].Welding_Pos.Z=Lin_Pos.Z
N225_Short_Craft[Work_Area,1].Welding_Pos.A=Lin_Pos.A
N225_Short_Craft[Work_Area,1].Welding_Pos.B=Lin_Pos.B
N225_Short_Craft[Work_Area,1].Welding_Pos.C=Lin_Pos.C

CASE 2
SWITCH Sink_Welding_Size.Sink_Type
CASE #UpDown_One

Lin_Pos.X=D225_Start_POS.X
Lin_Pos.Y=D225_Start_POS.Y

;Lin_Pos.X=0
;Lin_Pos.Y=Sink_Welding_Size.Sink_Size_Short_OnePos+Sink_Welding_Size.Sink_Size_Short_TwoPos
Lin_Pos.Z=0
Lin_Pos.A=0
Lin_Pos.B=0
Lin_Pos.C=0
case #LeftRight_One

Lin_Pos.X=D225_Start_POS.X
Lin_Pos.Y=D225_Start_POS.Y

;Lin_Pos.X=Sink_Welding_Size.Sink_Size_Short_OnePos
;Lin_Pos.Y=Sink_Welding_Size.Sink_Size_Long+Sink_Welding_Size.Sink_Size_Left_Distance*2
Lin_Pos.Z=0
Lin_Pos.A=0
Lin_Pos.B=0
Lin_Pos.C=0
ENDSWITCH


N225_Short_Craft[Work_Area,2].Welding_Pos.X=Lin_Pos.X
N225_Short_Craft[Work_Area,2].Welding_Pos.Y=Lin_Pos.Y
N225_Short_Craft[Work_Area,2].Welding_Pos.Z=Lin_Pos.Z
N225_Short_Craft[Work_Area,2].Welding_Pos.A=Lin_Pos.A
N225_Short_Craft[Work_Area,2].Welding_Pos.B=Lin_Pos.B
N225_Short_Craft[Work_Area,2].Welding_Pos.C=Lin_Pos.C

CASE 3
SWITCH Sink_Welding_Size.Sink_Type
CASE #UpDown_One


Lin_Pos.X=D225_End_POS.X
Lin_Pos.Y=D225_End_POS.Y

;Lin_Pos.X=Sink_Welding_Size.Sink_Size_Short_Side
;Lin_Pos.Y=Sink_Welding_Size.Sink_Size_Short_OnePos+Sink_Welding_Size.Sink_Size_Short_TwoPos
Lin_Pos.Z=0
Lin_Pos.A=0
Lin_Pos.B=0
Lin_Pos.C=0
case #LeftRight_One

Lin_Pos.X=D225_End_POS.X
Lin_Pos.Y=D225_End_POS.Y

;Lin_Pos.X=Sink_Welding_Size.Sink_Size_Short_OnePos
;Lin_Pos.Y=Sink_Welding_Size.Sink_Size_Long+Sink_Welding_Size.Sink_Size_Left_Distance*2-Sink_Welding_Size.Sink_Size_Short_Side
Lin_Pos.Z=0
Lin_Pos.A=0
Lin_Pos.B=0
Lin_Pos.C=0
ENDSWITCH


N225_Short_Craft[Work_Area,3].Welding_Pos.X=Lin_Pos.X
N225_Short_Craft[Work_Area,3].Welding_Pos.Y=Lin_Pos.Y
N225_Short_Craft[Work_Area,3].Welding_Pos.Z=Lin_Pos.Z
N225_Short_Craft[Work_Area,3].Welding_Pos.A=Lin_Pos.A
N225_Short_Craft[Work_Area,3].Welding_Pos.B=Lin_Pos.B
N225_Short_Craft[Work_Area,3].Welding_Pos.C=Lin_Pos.C

CASE 4
SWITCH Sink_Welding_Size.Sink_Type
CASE #UpDown_One

UL_Equation(D225_Start_POS,D225_End_POS,(Surr_Path*0.01),Sink_Welding_Size.Sink_Size_R,Lin_Pos)

;Lin_Pos.X=Sink_Welding_Size.Sink_Size_Short_Side-Sink_Welding_Size.Sink_Size_Short_Side*(Surr_Path/100)
;Lin_Pos.Y=Sink_Welding_Size.Sink_Size_Short_OnePos+Sink_Welding_Size.Sink_Size_Short_TwoPos
Lin_Pos.Z=-150.000
Lin_Pos.A=0
Lin_Pos.B=0
Lin_Pos.C=0
case #LeftRight_One

UL_Equation(D225_Start_POS,D225_End_POS,(Surr_Path*0.01),Sink_Welding_Size.Sink_Size_R,Lin_Pos)

;Lin_Pos.X=Sink_Welding_Size.Sink_Size_Short_OnePos
;Lin_Pos.Y=Sink_Welding_Size.Sink_Size_Long+Sink_Welding_Size.Sink_Size_Left_Distance+Sink_Welding_Size.Sink_Size_Short_Side*(Surr_Path/100)
Lin_Pos.Z=-150.000
Lin_Pos.A=0
Lin_Pos.B=0
Lin_Pos.C=0
ENDSWITCH


N225_Short_Craft[Work_Area,4].Welding_Pos.X=Lin_Pos.X
N225_Short_Craft[Work_Area,4].Welding_Pos.Y=Lin_Pos.Y
N225_Short_Craft[Work_Area,4].Welding_Pos.Z=Lin_Pos.Z
N225_Short_Craft[Work_Area,4].Welding_Pos.A=Lin_Pos.A
N225_Short_Craft[Work_Area,4].Welding_Pos.B=Lin_Pos.B
N225_Short_Craft[Work_Area,4].Welding_Pos.C=Lin_Pos.C

ENDSWITCH


CASE #N315
;
SWITCH  Offset_No

CASE 1
SWITCH Sink_Welding_Size.Sink_Type
CASE #UpDown_One

Lin_Pos.X=D315_Start_POS.X
Lin_Pos.Y=D315_Start_POS.Y


;Lin_Pos.X=Sink_Welding_Size.Sink_Size_Width+Sink_Welding_Size.Sink_Size_Down_Distance*2
;Lin_Pos.Y=Sink_Welding_Size.Sink_Size_Short_OnePos+Sink_Welding_Size.Sink_Size_Short_TwoPos
Lin_Pos.Z=-150.000
Lin_Pos.A=0
Lin_Pos.B=0
Lin_Pos.C=0

case #LeftRight_One


Lin_Pos.X=D315_Start_POS.X
Lin_Pos.Y=D315_Start_POS.Y

;Lin_Pos.X=Sink_Welding_Size.Sink_Size_Short_OnePos+Sink_Welding_Size.Sink_Size_Short_TwoPos
;Lin_Pos.Y=Sink_Welding_Size.Sink_Size_Long+Sink_Welding_Size.Sink_Size_Left_Distance*2
Lin_Pos.Z=-150.000
Lin_Pos.A=0
Lin_Pos.B=0
Lin_Pos.C=0
ENDSWITCH


N315_Short_Craft[Work_Area,1].Welding_Pos.X=Lin_Pos.X
N315_Short_Craft[Work_Area,1].Welding_Pos.Y=Lin_Pos.Y
N315_Short_Craft[Work_Area,1].Welding_Pos.Z=Lin_Pos.Z
N315_Short_Craft[Work_Area,1].Welding_Pos.A=Lin_Pos.A
N315_Short_Craft[Work_Area,1].Welding_Pos.B=Lin_Pos.B
N315_Short_Craft[Work_Area,1].Welding_Pos.C=Lin_Pos.C

CASE 2
SWITCH Sink_Welding_Size.Sink_Type
CASE #UpDown_One

Lin_Pos.X=D315_Start_POS.X
Lin_Pos.Y=D315_Start_POS.Y

;Lin_Pos.X=Sink_Welding_Size.Sink_Size_Width+Sink_Welding_Size.Sink_Size_Down_Distance*2
;Lin_Pos.Y=Sink_Welding_Size.Sink_Size_Short_OnePos+Sink_Welding_Size.Sink_Size_Short_TwoPos
Lin_Pos.Z=0
Lin_Pos.A=0
Lin_Pos.B=0
Lin_Pos.C=0

case #LeftRight_One

Lin_Pos.X=D315_Start_POS.X
Lin_Pos.Y=D315_Start_POS.Y


;Lin_Pos.X=Sink_Welding_Size.Sink_Size_Short_OnePos+Sink_Welding_Size.Sink_Size_Short_TwoPos
;Lin_Pos.Y=Sink_Welding_Size.Sink_Size_Long+Sink_Welding_Size.Sink_Size_Left_Distance*2
Lin_Pos.Z=0
Lin_Pos.A=0
Lin_Pos.B=0
Lin_Pos.C=0
ENDSWITCH


N315_Short_Craft[Work_Area,2].Welding_Pos.X=Lin_Pos.X
N315_Short_Craft[Work_Area,2].Welding_Pos.Y=Lin_Pos.Y
N315_Short_Craft[Work_Area,2].Welding_Pos.Z=Lin_Pos.Z
N315_Short_Craft[Work_Area,2].Welding_Pos.A=Lin_Pos.A
N315_Short_Craft[Work_Area,2].Welding_Pos.B=Lin_Pos.B
N315_Short_Craft[Work_Area,2].Welding_Pos.C=Lin_Pos.C

CASE 3
SWITCH Sink_Welding_Size.Sink_Type
CASE #UpDown_One

Lin_Pos.X=D315_End_POS.X
Lin_Pos.Y=D315_End_POS.Y


;Lin_Pos.X=Sink_Welding_Size.Sink_Size_Width+Sink_Welding_Size.Sink_Size_Down_Distance*2-Sink_Welding_Size.Sink_Size_Short_Side
;Lin_Pos.Y=Sink_Welding_Size.Sink_Size_Short_OnePos+Sink_Welding_Size.Sink_Size_Short_TwoPos
Lin_Pos.Z=0
Lin_Pos.A=0
Lin_Pos.B=0
Lin_Pos.C=0

case #LeftRight_One

Lin_Pos.X=D315_End_POS.X
Lin_Pos.Y=D315_End_POS.Y

;Lin_Pos.X=Sink_Welding_Size.Sink_Size_Short_OnePos+Sink_Welding_Size.Sink_Size_Short_TwoPos
;Lin_Pos.Y=Sink_Welding_Size.Sink_Size_Long+Sink_Welding_Size.Sink_Size_Left_Distance*2-Sink_Welding_Size.Sink_Size_Short_Side
Lin_Pos.Z=0
Lin_Pos.A=0
Lin_Pos.B=0
Lin_Pos.C=0
ENDSWITCH


N315_Short_Craft[Work_Area,3].Welding_Pos.X=Lin_Pos.X
N315_Short_Craft[Work_Area,3].Welding_Pos.Y=Lin_Pos.Y
N315_Short_Craft[Work_Area,3].Welding_Pos.Z=Lin_Pos.Z
N315_Short_Craft[Work_Area,3].Welding_Pos.A=Lin_Pos.A
N315_Short_Craft[Work_Area,3].Welding_Pos.B=Lin_Pos.B
N315_Short_Craft[Work_Area,3].Welding_Pos.C=Lin_Pos.C

CASE 4
SWITCH Sink_Welding_Size.Sink_Type
CASE #UpDown_One


UL_Equation(D315_Start_POS,D315_End_POS,(Surr_Path*0.01),Sink_Welding_Size.Sink_Size_R,Lin_Pos)

;Lin_Pos.X=Sink_Welding_Size.Sink_Size_Width+Sink_Welding_Size.Sink_Size_Down_Distance+Sink_Welding_Size.Sink_Size_Short_Side*(Surr_Path/100)
;Lin_Pos.Y=Sink_Welding_Size.Sink_Size_Short_OnePos+Sink_Welding_Size.Sink_Size_Short_TwoPos
Lin_Pos.Z=-150.000
Lin_Pos.A=0
Lin_Pos.B=0
Lin_Pos.C=0

case #LeftRight_One

UL_Equation(D315_Start_POS,D315_End_POS,(Surr_Path*0.01),Sink_Welding_Size.Sink_Size_R,Lin_Pos)

;Lin_Pos.X=Sink_Welding_Size.Sink_Size_Short_OnePos+Sink_Welding_Size.Sink_Size_Short_TwoPos
;Lin_Pos.Y=Sink_Welding_Size.Sink_Size_Long+Sink_Welding_Size.Sink_Size_Left_Distance+Sink_Welding_Size.Sink_Size_Short_Side*(Surr_Path/100)
Lin_Pos.Z=-150.000
Lin_Pos.A=0
Lin_Pos.B=0
Lin_Pos.C=0
ENDSWITCH

N315_Short_Craft[Work_Area,4].Welding_Pos.X=Lin_Pos.X
N315_Short_Craft[Work_Area,4].Welding_Pos.Y=Lin_Pos.Y
N315_Short_Craft[Work_Area,4].Welding_Pos.Z=Lin_Pos.Z
N315_Short_Craft[Work_Area,4].Welding_Pos.A=Lin_Pos.A
N315_Short_Craft[Work_Area,4].Welding_Pos.B=Lin_Pos.B
N315_Short_Craft[Work_Area,4].Welding_Pos.C=Lin_Pos.C
ENDSWITCH


ENDSWITCH

SWITCH Pos_Type

CASE #L_LIN_POS,#C_LIN_POS




Lin_Pos.X=Lin_Pos.X+Offset_info.X
Lin_Pos.Y=Lin_Pos.Y+Offset_info.Y
Lin_Pos.Z=Lin_Pos.Z+Offset_info.Z



CASE #C_CIR_POS





Cir_Middle_POS.X=Cir_Middle_POS.X+Offset_info.X
Cir_Middle_POS.Y=Cir_Middle_POS.Y+Offset_info.Y
Cir_Middle_POS.Z=Cir_Middle_POS.Z+Offset_info.Z

Cir_END_POS.X=Cir_END_POS.X+Offset_cir_info.X
Cir_END_POS.Y=Cir_END_POS.Y+Offset_cir_info.Y
Cir_END_POS.Z=Cir_END_POS.Z+Offset_cir_info.Z

ENDSWITCH


END

GLOBAL DEF HanGao_Camera_Offset(Vision_Model:IN ,Calibration_Area:IN,Work_Camera:IN, OFFSET_POS:OUT)
DECL E6POS OFFSET_POS,Cam_45_POS,Cam_135_POS,Cam_225_POS,Cam_315_POS
DECL INT Calibration_Area,Work_Camera
DECL Surround_Welding_Type Sink_Size
DECL REAL T_X,T_Y,Q_X,Q_Y
DECL Vision_Model_Enum Vision_Model



switch Work_Camera

CASE 1

Sink_Size=N1_Sink_Data
Cam_45_POS=N1_Cam_45_POS
Cam_135_POS=N1_Cam_135_POS
Cam_225_POS=N1_Cam_225_POS
Cam_315_POS=N1_Cam_315_POS

CASE 2
Sink_Size=N2_Sink_Data
Cam_45_POS=N2_Cam_45_POS
Cam_135_POS=N2_Cam_135_POS
Cam_225_POS=N2_Cam_225_POS
Cam_315_POS=N2_Cam_315_POS

ENDSWITCH



SWITCH Calibration_Area

CASE 1


Q_Y=Camera_Calibration_Data.Sink_Size_Left_Distance-Sink_Size.Sink_Size_Left_Distance
Q_X=(Camera_Calibration_Data.Sink_Size_Down_Distance+Camera_Calibration_Data.Sink_Size_Width)-(Sink_Size.Sink_Size_Down_Distance+Sink_Size.Sink_Size_Width)

SWITCH Vision_Model

case #Calibration

IF (ABS(Q_Y)>=Vision_Scope ) OR (ABS(Q_X)>=Vision_Scope)THEN

OFFSET_POS=Cam_45_POS
OFFSET_POS.X=Cam_45_POS.X-Q_X
OFFSET_POS.Y=Cam_45_POS.Y-Q_Y

ELSE
OFFSET_POS=Cam_45_POS

ENDIF

ENDSWITCH

CASE 2


Q_Y=Camera_Calibration_Data.Sink_Size_Left_Distance-Sink_Size.Sink_Size_Left_Distance
Q_X=Camera_Calibration_Data.Sink_Size_Down_Distance-Sink_Size.Sink_Size_Down_Distance


SWITCH Vision_Model

case #Calibration
IF (ABS(Q_Y)>=Vision_Scope ) OR (ABS(Q_X)>=Vision_Scope)THEN
OFFSET_POS=Cam_135_POS
OFFSET_POS.X=Cam_135_POS.X-Q_X
OFFSET_POS.Y=Cam_135_POS.Y-Q_Y
ELSE
OFFSET_POS=Cam_135_POS

ENDIF

ENDSWITCH


CASE 3

Q_Y=(Camera_Calibration_Data.Sink_Size_Left_Distance+Camera_Calibration_Data.Sink_Size_Long)  -(Sink_Size.Sink_Size_Left_Distance+Sink_Size.Sink_Size_Long)
Q_X=Camera_Calibration_Data.Sink_Size_Down_Distance-Sink_Size.Sink_Size_Down_Distance

SWITCH Vision_Model

case #Calibration

IF (ABS(Q_Y)>=Vision_Scope ) OR (ABS(Q_X)>=Vision_Scope)THEN
OFFSET_POS=Cam_225_POS
OFFSET_POS.X=Cam_225_POS.X-Q_X
OFFSET_POS.Y=Cam_225_POS.Y-Q_Y
ELSE
OFFSET_POS=Cam_225_POS

ENDIF

ENDSWITCH


CASE 4

Q_Y=(Camera_Calibration_Data.Sink_Size_Left_Distance+Camera_Calibration_Data.Sink_Size_Long)-(Sink_Size.Sink_Size_Left_Distance+Sink_Size.Sink_Size_Long)
Q_X=(Camera_Calibration_Data.Sink_Size_Down_Distance+Camera_Calibration_Data.Sink_Size_Width)-(Sink_Size.Sink_Size_Down_Distance+Sink_Size.Sink_Size_Width)

SWITCH Vision_Model

case #Calibration
IF (ABS(Q_Y)>=Vision_Scope ) OR (ABS(Q_X)>=Vision_Scope)THEN
OFFSET_POS=Cam_315_POS
OFFSET_POS.X=Cam_315_POS.X-Q_X
OFFSET_POS.Y=Cam_315_POS.Y-Q_Y
ELSE
OFFSET_POS=Cam_315_POS

ENDIF

ENDSWITCH


ENDSWITCH


SWITCH Vision_Model

case #Find_Model
IF (ABS(Q_Y)>=Vision_Scope ) OR (ABS(Q_X)>=Vision_Scope)THEN
OFFSET_POS.X=OFFSET_POS.X-Q_X
OFFSET_POS.Y=OFFSET_POS.Y-Q_Y
ENDIF
ENDSWITCH





END


GLOBAL DEF HanGao_Calibration_Point(Calibration_POS:OUT,Calib_NO:IN)
DECL E6POS Calibration_POS
DECL INT Calib_NO



switch Global_Calib_Model

Case #New

Calibration_Point[Calib_NO]=Calibration_POS

Case #Add


Case #Text

Calibration_POS.X=Calibration_Text[Calib_NO].X
Calibration_POS.Y=Calibration_Text[Calib_NO].Y
endswitch


END

GLOBAL DEF HanGao_Camera_Sink_Pos( Calibration_POS:out,Calibration:IN,Work_Camera:IN)
DECL INT Calibration,Work_Camera
DECL BOOL User_Revise
DECL CHAR Meg_Str[1024]
DECL Surround_Welding_Type Sink_Size
DECL E6POS Calibration_POS
 Meg_Str[]="This operation will overwrite the original data, whether to confirm?"
 ;Global_Messages_Dlg( Meg_Str[] ,User_Revise)
User_Revise=FALSE






switch Work_Camera

CASE 1

Sink_Size=N1_Sink_Data


SWITCH  Global_Calib_Model
CASE #Text

SWITCH Calibration
CASE 1
Calibration_POS=N1_Cam_45_POS
CASE 2
Calibration_POS=N1_Cam_135_POS
CASE 3
Calibration_POS=N1_Cam_225_POS
CASE 4
Calibration_POS=N1_Cam_315_POS
ENDSWITCH


CASE #New


Global_Messages_Dlg( Meg_Str[] ,User_Revise)
IF User_Revise==TRUE THEN

SWITCH Calibration
CASE 1
N1_Cam_45_POS=Calibration_POS
CASE 2
N1_Cam_135_POS=Calibration_POS
CASE 3
N1_Cam_225_POS=Calibration_POS
CASE 4
N1_Cam_315_POS=Calibration_POS
ENDSWITCH


Camera_Calibration_Data=Sink_Size
endif


ENDSWITCH


CASE 2

Sink_Size=N2_Sink_Data
SWITCH  Global_Calib_Model
CASE #Text

SWITCH Calibration
CASE 1
Calibration_POS=N2_Cam_45_POS
CASE 2
Calibration_POS=N2_Cam_135_POS
CASE 3
Calibration_POS=N2_Cam_225_POS
CASE 4
Calibration_POS=N2_Cam_315_POS
ENDSWITCH


CASE #New

Global_Messages_Dlg( Meg_Str[] ,User_Revise)
IF User_Revise==TRUE THEN

SWITCH Calibration
CASE 1
N2_Cam_45_POS=Calibration_POS
CASE 2
N2_Cam_135_POS=Calibration_POS
CASE 3
N2_Cam_225_POS=Calibration_POS
CASE 4
N2_Cam_315_POS=Calibration_POS
ENDSWITCH

Camera_Calibration_Data=Sink_Size

endif
ENDSWITCH

ENDSWITCH










END


GLOBAL DEF HanGao_Base_Calculate(POS_1:IN,POS_2:IN,POS_3:IN,POS_4:IN,G_BASE:IN,Angle_Area:IN)
DECL E6POS POS_1
DECL E6POS POS_2
DECL E6POS POS_3
DECL E6POS POS_4
DECL Work_Area_Enum Angle_Area
DECL REAL Direction_Deg,ATan_Deg
DECL INT G_BASE,OPFFSET
DECL Calculate_Lin_Const Lin_1_CONST
DECL Calculate_Lin_Const Lin_2_CONST
DECL POS Lin_Curss
DECL CHAR Meg_Str[1024]
DECL BOOL User_Revise
DECL State_t _State
SWRITE( Meg_Str[] , _State , OPFFSET , "New_BASE[%d]=X:%7.3F,Y:%7.3F,Z:%7.3F,A:%7.3F,B:%7.3F,C:%7.3F" , G_BASE ,Lin_Curss.X,Lin_Curss.Y,Lin_Curss.Z,Lin_Curss.A,Lin_Curss.B,Lin_Curss.C)



OPFFSET=0
Lin_Curss={X 0, Y 0, Z 0, A 0,B 0,C 0}




Lin_1_CONST.A=POS_2.Y-POS_1.Y
Lin_1_CONST.B=POS_1.X-POS_2.X
Lin_1_CONST.C=POS_2.X*POS_1.Y-POS_1.X*POS_2.Y

Lin_2_CONST.A=POS_4.Y-POS_3.Y
Lin_2_CONST.B=POS_3.X-POS_4.X
Lin_2_CONST.C=POS_4.X*POS_3.Y-POS_3.X*POS_4.Y


Lin_Curss.X=(Lin_1_CONST.B*Lin_2_CONST.C-Lin_2_CONST.B*Lin_1_CONST.C)/(Lin_1_CONST.A*Lin_2_CONST.B-Lin_2_CONST.A*Lin_1_CONST.B)
Lin_Curss.Y=(Lin_2_CONST.A*Lin_1_CONST.C-Lin_1_CONST.A*Lin_2_CONST.C)/(Lin_2_CONST.B*Lin_1_CONST.A-Lin_1_CONST.B*Lin_2_CONST.A)
Lin_Curss.Z=POS_1.Z



SWITCH Angle_Area


CASE #A0

Direction_Deg=-180.000

IF Lin_Curss.X<>POS_4.X THEN

ATan_Deg=ATAN2(ABS(POS_4.x-Lin_Curss.x),ABS(POS_4.y-Lin_Curss.y))

IF POS_4.X-Lin_Curss.X<0 THEN
Lin_Curss.A=Direction_Deg+ATan_Deg
ENDIF

IF POS_4.X-Lin_Curss.X>0 THEN
Lin_Curss.A=Direction_Deg-ATan_Deg
ENDIF


ELSE

Lin_Curss.A=Direction_Deg

ENDIF

CASE #A90

Direction_Deg=90.000

IF Lin_Curss.Y<>POS_4.Y THEN

ATan_Deg=ATAN2(ABS(POS_4.Y-Lin_Curss.Y),ABS(POS_4.X-Lin_Curss.X))

IF POS_4.Y-Lin_Curss.Y<0 THEN
Lin_Curss.A=Direction_Deg-ATan_Deg
ENDIF

IF POS_4.Y-Lin_Curss.Y>0 THEN
Lin_Curss.A=Direction_Deg+ATan_Deg
ENDIF


ELSE

Lin_Curss.A=Direction_Deg

ENDIF




CASE #A270

Direction_Deg=-90.000

IF Lin_Curss.Y<>POS_4.Y THEN

ATan_Deg=ATAN2(ABS(POS_4.Y-Lin_Curss.Y),ABS(POS_4.X-Lin_Curss.X))

IF POS_4.Y-Lin_Curss.Y<0 THEN
Lin_Curss.A=Direction_Deg+ATan_Deg
ENDIF

IF POS_4.Y-Lin_Curss.Y>0 THEN
Lin_Curss.A=Direction_Deg-ATan_Deg
ENDIF


ELSE

Lin_Curss.A=Direction_Deg

ENDIF




ENDSWITCH










Lin_Curss.B=0
Lin_Curss.C=-180.000


SWRITE( Meg_Str[] , _State , OPFFSET , "New_BASE[%d]=X:%7.3F,Y:%7.3F,Z:%7.3F,A:%7.3F,B:%7.3F,C:%7.3F" , G_BASE ,Lin_Curss.X,Lin_Curss.Y,Lin_Curss.Z,Lin_Curss.A,Lin_Curss.B,Lin_Curss.C)


Global_Messages_Dlg( Meg_Str[] ,User_Revise)

IF User_Revise==TRUE THEN

IF G_BASE<>0  THEN

BASE_DATA[G_BASE].X=Lin_Curss.X
BASE_DATA[G_BASE].Y=Lin_Curss.Y
BASE_DATA[G_BASE].Z=Lin_Curss.Z
BASE_DATA[G_BASE].A=Lin_Curss.A
BASE_DATA[G_BASE].B=Lin_Curss.B
BASE_DATA[G_BASE].C=Lin_Curss.C

ENDIF

ENDIF


END


GLobAL DEF HanGao_DAT_ACT( Weld_Dat:IN,Weld_LDAT:IN)
DECL Surr_Welding_Craft_Type Weld_DAT
DECL LDAT Weld_LDAT


TRIGGER WHEN PATH=0 DELAY=0 DO $ANOUT[1]=Weld_Dat.Welding_Power/100
Weld_LDAT.VEL=Weld_Dat.Welding_Speed
Weld_LDAT.ACC=Weld_Dat.Welding_ACC
Weld_LDAT.APO_DIST=Weld_Dat.Welding_CDIS



END


GLOBAL DEF Global_Messages_Dlg( Messsage_All[]:IN , User_S:OUT)

DECL KrlMsg_T msg
DECL KrlMsgPar_T Par[3]
DECL KrlmsgOpt_T opt
DECL KrlMsgDlgSK_T SK[7]
DECL INT nHandle,keynumber,OPFFSET
DECl BOOL User_S
DECL CHAR Messsage_All[]



msg={modul[] "HanGao" ,Nr 7}
msg.msg_txt[] = Messsage_All[]
SK[1]={sk_Type #value, sk_txt[] "Yes"}
SK[2]={sk_type #value, sk_txt[] "NO" }

nHandle= Set_KrlDlg( msg, par[],sk[],opt)

IF (nHandle>0) THEN

While (Exists_KrlDlg(nHandle,keynumber))
 wait sec 0.1
ENDWhile

SWITCH keynumber
   case 1
   User_S=true

   case 2
   User_S=false

ENDSWITCH










ENDIF


END


;Ax+By+C=0
GLOBAL DEF Lin_Equation (P1:IN,P2:IN,L_A:OUT,L_B:OUT,L_C:OUT)
DECL E6POS P1,P2
DECL REAL A,B,C,L_A,L_B,L_C
L_A=0.00
L_B=0.00
L_C=0.00



L_A=P2.Y-P1.Y
L_B=P1.X-P2.X
L_C=P2.X*P1.Y-P1.X*P2.Y




END



;y=kx+b
GLOBAL DEF Lin_Equation_LTk (A:IN,B:IN,C:IN,K_K:OUT,K_B:OUT)
DECL REAL A,B,C,K_K,K_B
K_K=0
K_B=0

K_K=-(a/b)
K_B=-(c/b)



END

;Point-User distance
GLOBAL DEF UL_Equation (UP1:IN,UP2:IN,U_DIS:IN,C_L:IN, Result_Pos_1:OUT)
DECL E6POS UP1,UP2,Result_Pos_1,L_S,L_E
DECL REAL L_Distance,L_DIS_1,L_DIS_2,U_DIS,R_X,R_Y,C_L



PP_Equation(UP1,UP2,L_DIS_1)

L_S.X=C_L*(UP2.X-UP1.X)/L_DIS_1+UP1.X
L_S.Y=C_L*(UP2.Y-UP1.Y)/L_DIS_1+UP1.Y

L_E.X=(L_DIS_1-C_L)*(UP2.X-UP1.X)/L_DIS_1+UP1.X
L_E.Y=(L_DIS_1-C_L)*(UP2.Y-UP1.Y)/L_DIS_1+UP1.Y

PP_Equation(L_S,L_E,L_DIS_2)


Result_Pos_1.X=L_DIS_2*U_DIS*(L_E.X-L_S.X)/L_DIS_2+L_S.X
Result_Pos_1.Y=L_DIS_2*U_DIS*(L_E.Y-L_S.Y)/L_DIS_2+L_S.Y


; IF U_DIS>1 THEN

; Result_Pos_1.X=U_DIS*(UP2.X-UP1.X)/L_DIS+UP1.X
; Result_Pos_1.Y=U_DIS*(UP2.Y-UP1.Y)/L_DIS+UP1.Y

; ELSE

; Result_Pos_1.X=L_DIS*U_DIS*(UP2.X-UP1.X)/L_DIS+UP1.X
; Result_Pos_1.Y=L_DIS*U_DIS*(UP2.Y-UP1.Y)/L_DIS+UP1.Y

; ENDIF





END



;Point-Point distance
GLOBAL DEF PP_Equation (PP1:IN,PP2:IN,L_Distance:OUT)
DECL E6POS PP1,PP2
DECL REAL L_Distance


L_Distance=0



L_Distance=SQRT((PP2.X-PP1.X)*(PP2.X-PP1.X)+(PP2.Y-PP1.Y)*(PP2.Y-PP1.Y))



END

--- Glode_HanGao.dat ---
&ACCESS RVO4
&REL 506
&PARAM EDITMASK = *
&PARAM TEMPLATE = C:\KRC\Roboter\Template\vorgabe
&PARAM DISKPATH = KRC:\R1\Program\HG
DEFDAT  GLODE_HANGAO PUBLIC



GLOBAL BOOL EKI_Server_Ini=TRUE
GLOBAL BOOL EKI_Server_Open=TRUE
GLOBAL BOOL EKI_Server_Connect=TRUE
GLOBAL BOOL EKI_Server_Receive=FALSE
GLOBAL BOOL EKI_Server_Send=FALSE
GLOBAL BOOL EKI_Server_Reset=FALSE


;--------DECL_Enum---------------
GLOBAL ENUM Sink_Type_Enum UpDown_One,LeftRight_One,LeftRight_Two,Null
GLOBAL ENUM Area_Enum L0,C45,L90,C135,L180,C225,L270,C315,N45,N135,N225,N315
GLOBAL ENUM Pos_Type_Enum C_LIN_POS,C_CIR_POS,L_LIN_POS
GLOBAL ENUM Work_Area_Enum A0,A90,A270
GLOBAL ENUM Vision_Model_Enum Calibration,Find_Model
GLOBAL ENUM Vision_Type_Enum Vision_Run,Vision_No,Vision_Text
GLOBAL ENUM Vision_PATH_Enum X,Y,Z,XY,XZ,YZ,XYZ,XYZABC
;----------------------------------
;---DECL-STRUC-------------------------


GLOBAL STRUC Surround_Welding_Type BOOL Write_Status,REAL Sink_Size_Long,REAL Sink_Size_Width,REAL Sink_Size_R,REAL Sink_Size_Short_Side,REAL Sink_Size_Short_OnePos,REAL Sink_Size_Short_TwoPos,REAL Sink_Size_Pots_Thick,REAL Sink_Size_Panel_Thick,INT Sink_Model,REAL Sink_Size_Left_Distance,REAL Sink_Size_Down_Distance,Sink_Type_Enum Sink_Type
GLOBAL STRUC LSC_TOOL_TYP INT LSR_MAX_PWR,INT LSR_MIN_PWR,INT LSR_Prg,REAL SNSR_Prg,INT SNSR_State,REAL GAS_Pressure,INT LSR_Dly,INT GAS_Pre_Flow,INT GAS_Post_Flow
GLOBAL STRUC Offset_POS REAL X,REAL Y,REAL Z,REAL A,REAL B,REAL C
GLOBAL STRUC Offset_CIR REAL C_X,REAL C_Y,REAL C_Z,REAL C_A,REAL C_B,REAL C_C
GLOBAL STRUC Calculate_Lin_Const REAL A,REAL B,REAL C
GLOBAL STRUC Calibration_Sink_TYP REAL Long,REAL Width
GLOBAL STRUC Calibrate_Data BOOL Calibrate_State,INT Plan_Base_No,CHAR Calib_Pos_Name_1[20],CHAR Calib_Pos_Name_2[20],CHAR Calib_Pos_Name_3[20],CHAR Calib_Pos_Name_4[20],CHAR Calib_Pos_Name_5[20],CHAR Calib_Pos_Name_6[20],CHAR Calib_Pos_Name_7[20],CHAR Calib_Pos_Name_8[20],CHAR Calib_Pos_Name_9[20],CHAR Calib_Pos_Name_10[20]



GLOBAL STRUC Surr_Welding_Craft_Type CHAR Welding_Name[20],E6POS Welding_Pos,REAL Welding_Power,REAL Welding_Speed,REAL Welding_Angle,INT Welding_CDIS,INT Welding_ACC,Offset_POS Welding_Offset,Offset_CIR Welding_Offset_CIR



;-------------------------------------


;----------DECL_Value----------------------
DECL GLOBAL Surround_Welding_Type SW_DEFAULT={Sink_Size_Long 50.0000,Sink_Size_Width 345.000,Sink_Size_R 10.0000,Sink_Size_Pots_Thick 0.750000,Sink_Size_Panel_Thick 2.85000,Sink_Model 952154,Sink_Type #UpDown_One}
DECL GLOBAL LSC_TOOL_TYP LTDEFAULT={LSR_MAX_PWR 500,LSR_MIN_PWR 50,LSR_Prg 1,SNSR_Prg 1.00000,SNSR_State 0,GAS_Pressure 1.00000,LSR_Dly 100,GAS_Pre_Flow 0,GAS_Post_Flow 0}
DECL GLOBAL Offset_POS FFDEFAULT={X 0.0,Y 0.0,Z 0.0,A 0.0,B 0.0,C 0.0}
DECL GLOBAL Offset_CIR FCDEFAULT={C_X 0.0,C_Y 0.0,C_Z 0.0,C_A 0.0,C_B 0.0,C_C 0.0}
DECL GLOBAL Calibrate_Data CDDEFAULT={Calibrate_State FALSE,Plan_Base_No 5,Calib_Pos_Name_1[] " ",Calib_Pos_Name_2[] " ",Calib_Pos_Name_3[] " ",Calib_Pos_Name_4[] " ",Calib_Pos_Name_5[] " ",Calib_Pos_Name_6[] " ",Calib_Pos_Name_7[] " ",Calib_Pos_Name_8[] " ",Calib_Pos_Name_9[] " ",Calib_Pos_Name_10[] " "}
DECL GLOBAL E6POS PODEFAULT={X 0.0,Y 0.0,Z 0.0,A 0.0,B 0.0,C 0.0}
DECL GLOBAL E6POS XDEFAULT={X 0.0,Y 0.0,Z 0.0,A 0.0,B 0.0,C 0.0,S 2,T 2,E1 0.0,E2 0.0,E3 0.0,E4 0.0,E5 0.0,E6 0.0}



DECL GLOBAL Surround_Welding_Type Camera_Calibration_Data={Sink_Size_Long 632.000,Sink_Size_Width 352.000,Sink_Size_R 10.0000,Sink_Size_Short_Side 23.0000,Sink_Size_Short_OnePos 36.0000,Sink_Size_Short_TwoPos 328.000,Sink_Size_Pots_Thick 0.0,Sink_Size_Panel_Thick 0.0,Sink_Model 952154,Sink_Size_Left_Distance 24.0000,Sink_Size_Down_Distance 24.0000,Sink_Type #LeftRight_One}

DECL GLOBAL E6POS N1_Cam_45_POS={X 293.000,Y 90.0000,Z -80.0000,A 0.0,B 0.0,C 0.0,S 2,T 10,E1 0.0,E2 0.0,E3 0.0,E4 0.0,E5 0.0,E6 0.0}
DECL GLOBAL E6POS N1_Cam_135_POS={X -42.0000,Y 90.0000,Z -80.0000,A 0.0,B 0.0,C 0.0,S 2,T 10,E1 0.0,E2 0.0,E3 0.0,E4 0.0,E5 0.0,E6 0.0}
DECL GLOBAL E6POS N1_Cam_225_POS={X -40.0000,Y 716.000,Z -80.0000,A 0.0,B 0.0,C 0.0,S 2,T 43,E1 0.0,E2 0.0,E3 0.0,E4 0.0,E5 0.0,E6 0.0}
DECL GLOBAL E6POS N1_Cam_315_POS={X 295.000,Y 714.000,Z -80.0000,A 0.0,B 0.0,C 0.0,S 2,T 43,E1 0.0,E2 0.0,E3 0.0,E4 0.0,E5 0.0,E6 0.0}

DECL GLOBAL E6POS N2_Cam_45_POS={X 293.122131,Y 89.9176636,Z -80.0293961,A 0.0,B 0.0,C 0.0,S 2,T 10,E1 0.0,E2 0.0,E3 0.0,E4 0.0,E5 0.0,E6 0.0}
DECL GLOBAL E6POS N2_Cam_135_POS={X -42.3839874,Y 91.8151550,Z -80.0254822,A 0.0,B 0.0,C 0.0,S 2,T 10,E1 0.0,E2 0.0,E3 0.0,E4 0.0,E5 0.0,E6 0.0}
DECL GLOBAL E6POS N2_Cam_225_POS={X -39.7999954,Y 716.082336,Z -80.0293350,A 0.0,B 0.0,C 0.0,S 2,T 43,E1 0.0,E2 0.0,E3 0.0,E4 0.0,E5 0.0,E6 0.0}
DECL GLOBAL E6POS N2_Cam_315_POS={X 294.984924,Y 714.198059,Z -80.0293350,A 0.0,B 0.0,C 0.0,S 2,T 43,E1 0.0,E2 0.0,E3 0.0,E4 0.0,E5 0.0,E6 0.0}

DECL GLOBAL E6POS N45_OFFSET_POS={X 375.888,Y 19.1080,Z 0.0,A 0.0,B 0.0,C 0.0}
DECL GLOBAL E6POS N135_OFFSET_POS={X 19.2480,Y 19.4280,Z 0.0,A 0.0,B 0.0,C 0.0}
DECL GLOBAL E6POS N225_OFFSET_POS={X 18.8370,Y 660.925,Z 0.0,A 0.0,B 0.0,C 0.0}
DECL GLOBAL E6POS N315_OFFSET_POS={X 375.531,Y 661.361,Z 0.0,A 0.0,B 0.0,C 0.0}

DECL GLOBAL E6POS N45_CIR_POS={X 370.887,Y 21.4200,Z 0.0,A 0.0,B 0.0,C 0.0}
DECL GLOBAL E6POS N135_CIR_POS={X 23.1220,Y 23.0800,Z 0.0,A 0.0,B 0.0,C 0.0}
DECL GLOBAL E6POS N225_CIR_POS={X 22.5580,Y 657.093,Z 0.0,A 0.0,B 0.0,C 0.0}
DECL GLOBAL E6POS N315_CIR_POS={X 371.252,Y 658.128,Z 0.0,A 0.0,B 0.0,C 0.0}

DECL GLOBAL E6POS D45_Start_POS={X 363.069,Y 0.172000,Z 0.0,A 0.0,B 0.0,C 0.0}
DECL GLOBAL E6POS D45_End_POS={X 363.226,Y 19.0740,Z 0.0,A 0.0,B 0.0,C 0.0}
DECL GLOBAL E6POS D135_Start_POS={X 31.9650,Y 0.265000,Z 0.0,A 0.0,B 0.0,C 0.0}
DECL GLOBAL E6POS D135_End_POS={X 31.7740,Y 19.3580,Z 0.0,A 0.0,B 0.0,C 0.0}
DECL GLOBAL E6POS D225_Start_POS={X 31.1060,Y 680.043,Z 0.0,A 0.0,B 0.0,C 0.0}
DECL GLOBAL E6POS D225_End_POS={X 30.9840,Y 660.897,Z 0.0,A 0.0,B 0.0,C 0.0}
DECL GLOBAL E6POS D315_Start_POS={X 363.308,Y 680.243,Z 0.0,A 0.0,B 0.0,C 0.0}
DECL GLOBAL E6POS D315_End_POS={X 363.008,Y 661.355,Z 0.0,A 0.0,B 0.0,C 0.0}


DECL GLOBAL Surr_Welding_Craft_Type L0_Welding_Craft[2,10]
L0_Welding_Craft[1,1]={Welding_Name[] "S2",Welding_Pos {X 375.389648,Y 92.3825073,Z 1.50000,A 0.0,B 20.0000,C 0.0},Welding_Power 58.0000,Welding_Speed 0.400000,Welding_Angle 20.0000,Welding_CDIS 5,Welding_ACC 100,Welding_Offset {X 0.0,Y 0.0,Z 0.0}}
L0_Welding_Craft[1,2]={Welding_Name[] "L0_S2",Welding_Pos {X 375.159363,Y 586.834473,Z 1.50000,A 0.0,B 20.0000,C 0.0},Welding_Power 58.0000,Welding_Speed 0.0450000,Welding_Angle 20.0000,Welding_CDIS 5,Welding_ACC 100,Welding_Offset {X -1.00000,Y 0.0,Z 0.0}}
L0_Welding_Craft[1,3]={Welding_Name[] "L0_S3",Welding_Pos {X 375.274506,Y 339.608490,Z 1.50000,A 0.0,B 20.0000,C 0.0},Welding_Power 58.0000,Welding_Speed 0.0450000,Welding_Angle 20.0000,Welding_CDIS 5,Welding_ACC 100,Welding_Offset {X -0.500000,Y 0.0,Z 0.0}}
L0_Welding_Craft[1,4]={Welding_Name[] "L0_S4",Welding_Pos {X 375.418427,Y 30.5759888,Z 1.50000,A 0.0,B 20.0000,C 0.0},Welding_Power 58.0000,Welding_Speed 0.0450000,Welding_Angle 20.0000,Welding_CDIS 5,Welding_ACC 100,Welding_Offset {X -0.500000,Y 0.0,Z 0.0}}
L0_Welding_Craft[1,5]={Welding_Name[] "S1",Welding_Pos {X 400.000,Y 86.0000153,Z -3.00000,A 0.0,B 23.0000,C 0.0},Welding_Power 80.0000,Welding_Speed 0.0400000,Welding_Angle 20.0000,Welding_CDIS 5,Welding_ACC 100,Welding_Offset {X 0.0,Y 0.0,Z 0.0}}
L0_Welding_Craft[1,6]={Welding_Name[] "S6",Welding_Pos {X 533.000,Y 463.600037,Z -2.05000,A 0.0,B -23.0000,C 0.0},Welding_Power 80.0000,Welding_Speed 0.0400000,Welding_Angle 20.0000,Welding_CDIS 5,Welding_ACC 100,Welding_Offset {X 0.0,Y 0.0,Z 0.0}}
L0_Welding_Craft[1,7]={Welding_Name[] "S7",Welding_Pos {X 533.000,Y 463.600037,Z -2.05000,A 0.0,B -23.0000,C 0.0},Welding_Power 80.0000,Welding_Speed 0.0400000,Welding_Angle 20.0000,Welding_CDIS 5,Welding_ACC 100,Welding_Offset {X 0.0,Y 0.0,Z 0.0}}
L0_Welding_Craft[1,8]={Welding_Name[] "S8",Welding_Pos {X 533.000,Y 463.600037,Z -2.05000,A 0.0,B -23.0000,C 0.0},Welding_Power 80.0000,Welding_Speed 0.0400000,Welding_Angle 20.0000,Welding_CDIS 5,Welding_ACC 100,Welding_Offset {X 0.0,Y 0.0,Z 0.0}}
L0_Welding_Craft[1,9]={Welding_Name[] "S9",Welding_Pos {X 533.000,Y 463.600037,Z -2.05000,A 0.0,B -23.0000,C 0.0},Welding_Power 80.0000,Welding_Speed 0.0400000,Welding_Angle 20.0000,Welding_CDIS 5,Welding_ACC 100,Welding_Offset {X 0.0,Y 0.0,Z 0.0}}
L0_Welding_Craft[1,10]={Welding_Name[] "S10",Welding_Pos {X 533.000,Y 338.000,Z -2.05000,A 0.0,B -23.0000,C 0.0},Welding_Power 80.0000,Welding_Speed 0.0400000,Welding_Angle 20.0000,Welding_CDIS 5,Welding_ACC 100,Welding_Offset {X 0.0,Y 0.0,Z 0.0}}
L0_Welding_Craft[2,1]={Welding_Name[] "L0_S1",Welding_Pos {X 375.846954,Y 92.9332886,Z 1.50000,A 0.0,B 20.0000,C 0.0},Welding_Power 60.0000,Welding_Speed 0.480000,Welding_Angle 20.0000,Welding_CDIS 0,Welding_ACC 100,Welding_Offset {X 0.100000,Y 0.0,Z 1.00000}}
L0_Welding_Craft[2,2]={Welding_Name[] "L0_S2",Welding_Pos {X 375.572052,Y 587.535706,Z 1.50000,A 0.0,B 20.0000,C 0.0},Welding_Power 60.0000,Welding_Speed 0.0450000,Welding_Angle 20.0000,Welding_CDIS 5,Welding_ACC 100,Welding_Offset {X -0.200000,Y 0.0,Z 1.00000}}
L0_Welding_Craft[2,3]={Welding_Name[] "L0_S3",Welding_Pos {X 375.709503,Y 340.234497,Z 1.50000,A 0.0,B 20.0000,C 0.0},Welding_Power 60.0000,Welding_Speed 0.0450000,Welding_Angle 20.0000,Welding_CDIS 5,Welding_ACC 100,Welding_Offset {X -0.300000,Y 0.0,Z 1.00000}}
L0_Welding_Craft[2,4]={Welding_Name[] "L0_S4",Welding_Pos {X 375.881317,Y 31.1079712,Z 1.50000,A 0.0,B 20.0000,C 0.0},Welding_Power 60.0000,Welding_Speed 0.0400000,Welding_Angle 20.0000,Welding_CDIS 5,Welding_ACC 100,Welding_Offset {X -0.200000,Y 0.0,Z 1.00000}}
L0_Welding_Craft[2,5]={Welding_Name[] "S1",Welding_Pos {X 400.000,Y 86.0000153,Z -3.00000,A 0.0,B 23.0000,C 0.0},Welding_Power 80.0000,Welding_Speed 0.0400000,Welding_Angle 20.0000,Welding_CDIS 5,Welding_ACC 100,Welding_Offset {X 0.0,Y 0.0,Z 0.0}}
L0_Welding_Craft[2,6]={Welding_Name[] "S6",Welding_Pos {X 533.000,Y 463.600037,Z -2.05000,A 0.0,B -23.0000,C 0.0},Welding_Power 80.0000,Welding_Speed 0.0400000,Welding_Angle 20.0000,Welding_CDIS 5,Welding_ACC 100,Welding_Offset {X 0.0,Y 0.0,Z 0.0}}
L0_Welding_Craft[2,7]={Welding_Name[] "S7",Welding_Pos {X 533.000,Y 463.600037,Z -2.05000,A 0.0,B -23.0000,C 0.0},Welding_Power 80.0000,Welding_Speed 0.0400000,Welding_Angle 20.0000,Welding_CDIS 5,Welding_ACC 100,Welding_Offset {X 0.0,Y 0.0,Z 0.0}}
L0_Welding_Craft[2,8]={Welding_Name[] "S8",Welding_Pos {X 533.000,Y 463.600037,Z -2.05000,A 0.0,B -23.0000,C 0.0},Welding_Power 80.0000,Welding_Speed 0.0400000,Welding_Angle 20.0000,Welding_CDIS 5,Welding_ACC 100,Welding_Offset {X 0.0,Y 0.0,Z 0.0}}
L0_Welding_Craft[2,9]={Welding_Name[] "S9",Welding_Pos {X 533.000,Y 463.600037,Z -2.05000,A 0.0,B -23.0000,C 0.0},Welding_Power 80.0000,Welding_Speed 0.0400000,Welding_Angle 20.0000,Welding_CDIS 5,Welding_ACC 100,Welding_Offset {X 0.0,Y 0.0,Z 0.0}}
L0_Welding_Craft[2,10]={Welding_Name[] "S10",Welding_Pos {X 533.000,Y 338.000,Z -2.05000,A 0.0,B -23.0000,C 0.0},Welding_Power 80.0000,Welding_Speed 0.0400000,Welding_Angle 20.0000,Welding_CDIS 5,Welding_ACC 100,Welding_Offset {X 0.0,Y 0.0,Z 0.0}}



DECL GLOBAL Surr_Welding_Craft_Type C45_Welding_Craft[2,3]
C45_Welding_Craft[1,1]={Welding_Name[] "C45_S1",Welding_Pos {X 375.418427,Y 30.5759888,Z 1.50000,A 0.0,B 20.0000,C 0.0},Welding_Power 80.0000,Welding_Speed 0.0400000,Welding_Angle 20.0000,Welding_CDIS 5,Welding_ACC 100,Welding_Offset {X 0.0,Y 0.0,Z -1.00000}}
C45_Welding_Craft[1,2]={Welding_Name[] "PM3",Welding_Pos {X 370.291,Y 20.8820,Z 1.50000,A 0.0,B 0.0,C 0.0},Welding_Power 80.0000,Welding_Speed 0.0400000,Welding_Angle 20.0000,Welding_CDIS 5,Welding_ACC 100,Welding_Offset {X 0.500000,Y 0.500000,Z -1.00000},Welding_Offset_CIR {C_X 0.0,C_Y 0.0,C_Z 0.0}}
C45_Welding_Craft[1,3]={Welding_Name[] "PE3",Welding_Pos {X 363.424,Y 18.5840397,Z 1.50000,A 0.0,B 0.0,C 20.0000},Welding_Power 58.0000,Welding_Speed 0.0200000,Welding_Angle 20.0000,Welding_CDIS 5,Welding_ACC 100,Welding_Offset {X 0.0,Y 0.0,Z -1.00000}}
C45_Welding_Craft[2,1]={Welding_Name[] "C45_S1",Welding_Pos {X 375.881317,Y 31.1079712,Z 1.50000,A 0.0,B 20.0000,C 0.0},Welding_Power 65.0000,Welding_Speed 0.0400000,Welding_Angle 20.0000,Welding_CDIS 40,Welding_ACC 80,Welding_Offset {X 0.0,Y 0.0,Z 0.0}}
C45_Welding_Craft[2,2]={Welding_Name[] "PM3",Welding_Pos {X 370.887,Y 21.4200,Z 1.50000,A 0.0,B 0.0,C 0.0},Welding_Power 60.0000,Welding_Speed 0.0400000,Welding_Angle 20.0000,Welding_CDIS 5,Welding_ACC 100,Welding_Offset {X 1.60000,Y 2.30000,Z 0.0},Welding_Offset_CIR {C_X 0.0,C_Y 0.0,C_Z 0.0}}
C45_Welding_Craft[2,3]={Welding_Name[] "PE3",Welding_Pos {X 363.888,Y 19.1187668,Z 1.50000,A 0.0,B 0.0,C 20.0000},Welding_Power 60.0000,Welding_Speed 0.0230000,Welding_Angle 20.0000,Welding_CDIS 5,Welding_ACC 100,Welding_Offset {X 0.0,Y 0.200000,Z 0.0}}


DECL GLOBAL Surr_Welding_Craft_Type L90_Welding_Craft[2,10]
L90_Welding_Craft[1,1]={Welding_Name[] "L90_S1",Welding_Pos {X 330.151611,Y 18.6063309,Z 1.50000,A 0.0,B 0.0,C 20.0000},Welding_Power 58.0000,Welding_Speed 0.0400000,Welding_Angle 20.0000,Welding_CDIS 5,Welding_ACC 100,Welding_Offset {X 0.0,Y 0.0,Z 0.0}}
L90_Welding_Craft[1,2]={Welding_Name[] "L90_S2",Welding_Pos {X 197.062012,Y 18.6955,Z 1.50000,A 0.0,B 0.0,C 20.0000},Welding_Power 58.0000,Welding_Speed 0.0400000,Welding_Angle 20.0000,Welding_CDIS 5,Welding_ACC 100,Welding_Offset {X 0.0,Y 0.0,Z 0.0}}
L90_Welding_Craft[1,3]={Welding_Name[] "L90_S3",Welding_Pos {X 63.9724121,Y 18.7846680,Z 1.50000,A 0.0,B 0.0,C 20.0000},Welding_Power 58.0000,Welding_Speed 0.0400000,Welding_Angle 20.0000,Welding_CDIS 5,Welding_ACC 100,Welding_Offset {X 0.0,Y -0.500000,Z 0.0}}
L90_Welding_Craft[1,4]={Welding_Name[] "S4",Welding_Pos {X 400.000,Y 86.0000153,Z -3.00000,A 0.0,B 23.0000,C 0.0},Welding_Power 80.0000,Welding_Speed 0.0400000,Welding_Angle 20.0000,Welding_CDIS 5,Welding_ACC 100,Welding_Offset {X 0.0,Y 0.0,Z 0.0}}
L90_Welding_Craft[1,5]={Welding_Name[] "S5",Welding_Pos {X 371.000,Y 0.0,Z -3.00000,A 0.0,B 0.0,C 23.0000},Welding_Power 80.0000,Welding_Speed 0.0400000,Welding_Angle 20.0000,Welding_CDIS 5,Welding_ACC 100,Welding_Offset {X 0.0,Y 0.0,Z 0.0}}
L90_Welding_Craft[1,6]={Welding_Name[] "S6",Welding_Pos {X 533.000,Y 463.600037,Z -2.05000,A 0.0,B -23.0000,C 0.0},Welding_Power 80.0000,Welding_Speed 0.0400000,Welding_Angle 20.0000,Welding_CDIS 5,Welding_ACC 100,Welding_Offset {X 0.0,Y 0.0,Z 0.0}}
L90_Welding_Craft[1,7]={Welding_Name[] "S7",Welding_Pos {X 533.000,Y 463.600037,Z -2.05000,A 0.0,B -23.0000,C 0.0},Welding_Power 80.0000,Welding_Speed 0.0400000,Welding_Angle 20.0000,Welding_CDIS 5,Welding_ACC 100,Welding_Offset {X 0.0,Y 0.0,Z 0.0}}
L90_Welding_Craft[1,8]={Welding_Name[] "S8",Welding_Pos {X 533.000,Y 463.600037,Z -2.05000,A 0.0,B -23.0000,C 0.0},Welding_Power 80.0000,Welding_Speed 0.0400000,Welding_Angle 20.0000,Welding_CDIS 5,Welding_ACC 100,Welding_Offset {X 0.0,Y 0.0,Z 0.0}}
L90_Welding_Craft[1,9]={Welding_Name[] "S9",Welding_Pos {X 533.000,Y 463.600037,Z -2.05000,A 0.0,B -23.0000,C 0.0},Welding_Power 80.0000,Welding_Speed 0.0400000,Welding_Angle 20.0000,Welding_CDIS 5,Welding_ACC 100,Welding_Offset {X 0.0,Y 0.0,Z 0.0}}
L90_Welding_Craft[1,10]={Welding_Name[] "S10",Welding_Pos {X 533.000,Y 338.000,Z -2.05000,A 0.0,B -23.0000,C 0.0},Welding_Power 80.0000,Welding_Speed 0.0400000,Welding_Angle 20.0000,Welding_CDIS 5,Welding_ACC 100,Welding_Offset {X 0.0,Y 0.0,Z 0.0}}
L90_Welding_Craft[2,1]={Welding_Name[] "L90_S1",Welding_Pos {X 330.624,Y 19.1486130,Z 1.50000,A 0.0,B 0.0,C 20.0000},Welding_Power 63.0000,Welding_Speed 0.0450000,Welding_Angle 20.0000,Welding_CDIS 5,Welding_ACC 100,Welding_Offset {X 0.0,Y 0.400000,Z 0.0}}
L90_Welding_Craft[2,2]={Welding_Name[] "L90_S2",Welding_Pos {X 197.568,Y 19.2680,Z 1.50000,A 0.0,B 0.0,C 20.0000},Welding_Power 63.0000,Welding_Speed 0.0450000,Welding_Angle 20.0000,Welding_CDIS 5,Welding_ACC 100,Welding_Offset {X 0.0,Y 0.0,Z 0.0}}
L90_Welding_Craft[2,3]={Welding_Name[] "L90_S3",Welding_Pos {X 64.5119934,Y 19.3873863,Z 1.50000,A 0.0,B 0.0,C 20.0000},Welding_Power 60.0000,Welding_Speed 0.0450000,Welding_Angle 20.0000,Welding_CDIS 5,Welding_ACC 100,Welding_Offset {X 0.0,Y -0.400000,Z 0.0}}
L90_Welding_Craft[2,4]={Welding_Name[] "S4",Welding_Pos {X 400.000,Y 86.0000153,Z -3.00000,A 0.0,B 23.0000,C 0.0},Welding_Power 80.0000,Welding_Speed 0.0430000,Welding_Angle 20.0000,Welding_CDIS 5,Welding_ACC 100,Welding_Offset {X 0.0,Y 0.0,Z 0.0}}
L90_Welding_Craft[2,5]={Welding_Name[] "S5",Welding_Pos {X 371.000,Y 0.0,Z -3.00000,A 0.0,B 0.0,C 23.0000},Welding_Power 80.0000,Welding_Speed 0.0400000,Welding_Angle 20.0000,Welding_CDIS 5,Welding_ACC 100,Welding_Offset {X 0.0,Y 0.0,Z 0.0}}
L90_Welding_Craft[2,6]={Welding_Name[] "S6",Welding_Pos {X 533.000,Y 463.600037,Z -2.05000,A 0.0,B -23.0000,C 0.0},Welding_Power 80.0000,Welding_Speed 0.0400000,Welding_Angle 20.0000,Welding_CDIS 5,Welding_ACC 100,Welding_Offset {X 0.0,Y 0.0,Z 0.0}}
L90_Welding_Craft[2,7]={Welding_Name[] "S7",Welding_Pos {X 533.000,Y 463.600037,Z -2.05000,A 0.0,B -23.0000,C 0.0},Welding_Power 80.0000,Welding_Speed 0.0400000,Welding_Angle 20.0000,Welding_CDIS 5,Welding_ACC 100,Welding_Offset {X 0.0,Y 0.0,Z 0.0}}
L90_Welding_Craft[2,8]={Welding_Name[] "S8",Welding_Pos {X 533.000,Y 463.600037,Z -2.05000,A 0.0,B -23.0000,C 0.0},Welding_Power 80.0000,Welding_Speed 0.0400000,Welding_Angle 20.0000,Welding_CDIS 5,Welding_ACC 100,Welding_Offset {X 0.0,Y 0.0,Z 0.0}}
L90_Welding_Craft[2,9]={Welding_Name[] "S9",Welding_Pos {X 533.000,Y 463.600037,Z -2.05000,A 0.0,B -23.0000,C 0.0},Welding_Power 80.0000,Welding_Speed 0.0400000,Welding_Angle 20.0000,Welding_CDIS 5,Welding_ACC 100,Welding_Offset {X 0.0,Y 0.0,Z 0.0}}
L90_Welding_Craft[2,10]={Welding_Name[] "S10",Welding_Pos {X 533.000,Y 338.000,Z -2.05000,A 0.0,B -23.0000,C 0.0},Welding_Power 80.0000,Welding_Speed 0.0400000,Welding_Angle 20.0000,Welding_CDIS 5,Welding_ACC 100,Welding_Offset {X 0.0,Y 0.0,Z 0.0}}

DECL GLOBAL Surr_Welding_Craft_Type C135_Welding_Craft[2,3]
C135_Welding_Craft[1,1]={Welding_Name[] "C135_S1",Welding_Pos {X 30.7000122,Y 18.8069611,Z 1.50000,A 0.0,B 0.0,C 20.0000},Welding_Power 80.0000,Welding_Speed 0.0400000,Welding_Angle 20.0000,Welding_CDIS 5,Welding_ACC 100,Welding_Offset {X 0.0,Y -0.500000,Z -1.00000}}
C135_Welding_Craft[1,2]={Welding_Name[] "PM4",Welding_Pos {X 21.8080,Y 22.4770,Z 1.50000,A 0.0,B 0.0,C 0.0},Welding_Power 80.0000,Welding_Speed 0.0400000,Welding_Angle -20.0000,Welding_CDIS 5,Welding_ACC 100,Welding_Offset {X -0.500000,Y -0.500000,Z -1.00000},Welding_Offset_CIR {C_X 0.0,C_Y 0.0,C_Z 0.0}}
C135_Welding_Craft[1,3]={Welding_Name[] "PE4",Welding_Pos {X 18.6979065,Y 30.8150,Z 1.50000,A 0.0,B -20.0000,C 0.0},Welding_Power 58.0000,Welding_Speed 0.0200000,Welding_Angle -20.0000,Welding_CDIS 5,Welding_ACC 100,Welding_Offset {X -0.500000,Y 0.0,Z -1.00000}}
C135_Welding_Craft[2,1]={Welding_Name[] "C135_S1",Welding_Pos {X 31.2479858,Y 19.4172325,Z 1.50000,A 0.0,B 0.0,C 20.0000},Welding_Power 60.0000,Welding_Speed 0.0400000,Welding_Angle 20.0000,Welding_CDIS 5,Welding_ACC 100,Welding_Offset {X 0.0,Y -0.300000,Z 0.0}}
C135_Welding_Craft[2,2]={Welding_Name[] "PM4",Welding_Pos {X 23.1220,Y 23.0800,Z 1.50000,A 0.0,B 0.0,C 0.0},Welding_Power 60.0000,Welding_Speed 0.0400000,Welding_Angle -20.0000,Welding_CDIS 5,Welding_ACC 100,Welding_Offset {X 0.0,Y -1.40000,Z 0.0},Welding_Offset_CIR {C_X 0.0,C_Y 0.0,C_Z 0.0}}
C135_Welding_Craft[2,3]={Welding_Name[] "PE4",Welding_Pos {X 19.2403107,Y 31.4279976,Z 1.50000,A 0.0,B -20.0000,C 0.0},Welding_Power 60.0000,Welding_Speed 0.0200000,Welding_Angle -20.0000,Welding_CDIS 5,Welding_ACC 100,Welding_Offset {X -0.500000,Y -0.300000,Z 0.0}}

DECL GLOBAL Surr_Welding_Craft_Type L180_Welding_Craft[2,10]
L180_Welding_Craft[1,1]={Welding_Name[] "L180_S1",Welding_Pos {X 18.6871262,Y 92.5788956,Z 1.50000,A 0.0,B -20.0000,C 0.0},Welding_Power 58.0000,Welding_Speed 0.0400000,Welding_Angle -20.0000,Welding_CDIS 5,Welding_ACC 100,Welding_Offset {X -0.500000,Y 0.0,Z 0.0}}
L180_Welding_Craft[1,2]={Welding_Name[] "L180_S2",Welding_Pos {X 18.6440010,Y 339.634491,Z 1.50000,A 0.0,B -20.0000,C 0.0},Welding_Power 58.0000,Welding_Speed 0.0400000,Welding_Angle -20.0000,Welding_CDIS 5,Welding_ACC 100,Welding_Offset {X -0.200000,Y 2.77555756E-17,Z 0.0}}
L180_Welding_Craft[1,3]={Welding_Name[] "L180_S3",Welding_Pos {X 18.5954838,Y 617.572,Z 1.50000,A 0.0,B -20.0000,C 0.0},Welding_Power 58.0000,Welding_Speed 0.0400000,Welding_Angle -20.0000,Welding_CDIS 5,Welding_ACC 100,Welding_Offset {X 0.0,Y 0.0,Z 0.0}}
L180_Welding_Craft[1,4]={Welding_Name[] "S4",Welding_Pos {X 400.000,Y 86.0000153,Z -3.00000,A 0.0,B 23.0000,C 0.0},Welding_Power 80.0000,Welding_Speed 0.0400000,Welding_Angle -20.0000,Welding_CDIS 5,Welding_ACC 100,Welding_Offset {X 0.0,Y 0.0,Z 0.0}}
L180_Welding_Craft[1,5]={Welding_Name[] "S5",Welding_Pos {X 0.0,Y 371.000,Z -3.00000,A 0.0,B -23.0000,C 0.0},Welding_Power 80.0000,Welding_Speed 0.0400000,Welding_Angle -20.0000,Welding_CDIS 5,Welding_ACC 100,Welding_Offset {X 0.0,Y 0.0,Z 0.0}}
L180_Welding_Craft[1,6]={Welding_Name[] "S6",Welding_Pos {X 533.000,Y 463.600037,Z -2.05000,A 0.0,B -23.0000,C 0.0},Welding_Power 80.0000,Welding_Speed 0.0400000,Welding_Angle -20.0000,Welding_CDIS 5,Welding_ACC 100,Welding_Offset {X 0.0,Y 0.0,Z 0.0}}
L180_Welding_Craft[1,7]={Welding_Name[] "S7",Welding_Pos {X 533.000,Y 463.600037,Z -2.05000,A 0.0,B -23.0000,C 0.0},Welding_Power 80.0000,Welding_Speed 0.0400000,Welding_Angle -20.0000,Welding_CDIS 5,Welding_ACC 100,Welding_Offset {X 0.0,Y 0.0,Z 0.0}}
L180_Welding_Craft[1,8]={Welding_Name[] "S8",Welding_Pos {X 533.000,Y 463.600037,Z -2.05000,A 0.0,B -23.0000,C 0.0},Welding_Power 80.0000,Welding_Speed 0.0400000,Welding_Angle -20.0000,Welding_CDIS 5,Welding_ACC 100,Welding_Offset {X 0.0,Y 0.0,Z 0.0}}
L180_Welding_Craft[1,9]={Welding_Name[] "S9",Welding_Pos {X 533.000,Y 463.600037,Z -2.05000,A 0.0,B -23.0000,C 0.0},Welding_Power 80.0000,Welding_Speed 0.0400000,Welding_Angle -20.0000,Welding_CDIS 5,Welding_ACC 100,Welding_Offset {X 0.0,Y 0.0,Z 0.0}}
L180_Welding_Craft[1,10]={Welding_Name[] "S10",Welding_Pos {X 533.000,Y 338.000,Z -2.05000,A 0.0,B -23.0000,C 0.0},Welding_Power 80.0000,Welding_Speed 0.0400000,Welding_Angle -20.0000,Welding_CDIS 5,Welding_ACC 100,Welding_Offset {X 0.0,Y 0.0,Z 0.0}}
L180_Welding_Craft[2,1]={Welding_Name[] "L180_S1",Welding_Pos {X 19.2007484,Y 93.1777,Z 1.50000,A 0.0,B -20.0000,C 0.0},Welding_Power 63.0000,Welding_Speed 0.0450000,Welding_Angle -20.0000,Welding_CDIS 5,Welding_ACC 100,Welding_Offset {X -0.700000,Y 0.0,Z 0.0}}
L180_Welding_Craft[2,2]={Welding_Name[] "L180_S2",Welding_Pos {X 19.0425,Y 340.176514,Z 1.50000,A 0.0,B -20.0000,C 0.0},Welding_Power 63.0000,Welding_Speed 0.0450000,Welding_Angle -20.0000,Welding_CDIS 5,Welding_ACC 100,Welding_Offset {X -0.300000,Y 0.0,Z 0.0}}
L180_Welding_Craft[2,3]={Welding_Name[] "L180_S3",Welding_Pos {X 18.8644695,Y 618.050110,Z 1.50000,A 0.0,B -20.0000,C 0.0},Welding_Power 63.0000,Welding_Speed 0.0450000,Welding_Angle -20.0000,Welding_CDIS 5,Welding_ACC 100,Welding_Offset {X -0.500000,Y 0.0,Z 0.0}}
L180_Welding_Craft[2,4]={Welding_Name[] "S4",Welding_Pos {X 400.000,Y 86.0000153,Z -3.00000,A 0.0,B 23.0000,C 0.0},Welding_Power 75.0000,Welding_Speed 0.0400000,Welding_Angle -20.0000,Welding_CDIS 5,Welding_ACC 100,Welding_Offset {X 0.0,Y 0.0,Z 0.0}}
L180_Welding_Craft[2,5]={Welding_Name[] "S5",Welding_Pos {X 0.0,Y 371.000,Z -3.00000,A 0.0,B -23.0000,C 0.0},Welding_Power 80.0000,Welding_Speed 0.0400000,Welding_Angle -20.0000,Welding_CDIS 5,Welding_ACC 100,Welding_Offset {X 0.0,Y 0.0,Z 0.0}}
L180_Welding_Craft[2,6]={Welding_Name[] "S6",Welding_Pos {X 533.000,Y 463.600037,Z -2.05000,A 0.0,B -23.0000,C 0.0},Welding_Power 80.0000,Welding_Speed 0.0400000,Welding_Angle -20.0000,Welding_CDIS 5,Welding_ACC 100,Welding_Offset {X 0.0,Y 0.0,Z 0.0}}
L180_Welding_Craft[2,7]={Welding_Name[] "S7",Welding_Pos {X 533.000,Y 463.600037,Z -2.05000,A 0.0,B -23.0000,C 0.0},Welding_Power 80.0000,Welding_Speed 0.0400000,Welding_Angle -20.0000,Welding_CDIS 5,Welding_ACC 100,Welding_Offset {X 0.0,Y 0.0,Z 0.0}}
L180_Welding_Craft[2,8]={Welding_Name[] "S8",Welding_Pos {X 533.000,Y 463.600037,Z -2.05000,A 0.0,B -23.0000,C 0.0},Welding_Power 80.0000,Welding_Speed 0.0400000,Welding_Angle -20.0000,Welding_CDIS 5,Welding_ACC 100,Welding_Offset {X 0.0,Y 0.0,Z 0.0}}
L180_Welding_Craft[2,9]={Welding_Name[] "S9",Welding_Pos {X 533.000,Y 463.600037,Z -2.05000,A 0.0,B -23.0000,C 0.0},Welding_Power 80.0000,Welding_Speed 0.0400000,Welding_Angle -20.0000,Welding_CDIS 5,Welding_ACC 100,Welding_Offset {X 0.0,Y 0.0,Z 0.0}}
L180_Welding_Craft[2,10]={Welding_Name[] "S10",Welding_Pos {X 533.000,Y 338.000,Z -2.05000,A 0.0,B -23.0000,C 0.0},Welding_Power 80.0000,Welding_Speed 0.0400000,Welding_Angle -20.0000,Welding_CDIS 5,Welding_ACC 100,Welding_Offset {X 0.0,Y 0.0,Z 0.0}}

DECL GLOBAL Surr_Welding_Craft_Type C225_Welding_Craft[2,3]
C225_Welding_Craft[1,1]={Welding_Name[] "C225_S1",Welding_Pos {X 18.5900936,Y 648.454,Z 1.50000,A 0.0,B -20.0000,C 0.0},Welding_Power 80.0000,Welding_Speed 0.0400000,Welding_Angle -20.0000,Welding_CDIS 5,Welding_ACC 100,Welding_Offset {X 0.0,Y 0.0,Z -1.00000}}
C225_Welding_Craft[1,2]={Welding_Name[] "PM5",Welding_Pos {X 22.1170,Y 656.630,Z 1.50000,A 0.0,B 0.0,C 0.0},Welding_Power 80.0000,Welding_Speed 0.0400000,Welding_Angle -20.0000,Welding_CDIS 5,Welding_ACC 100,Welding_Offset {X 0.500000,Y 0.500000,Z -1.00000},Welding_Offset_CIR {C_X 0.0,C_Y 0.0,C_Z 0.0}}
C225_Welding_Craft[1,3]={Welding_Name[] "PE5",Welding_Pos {X 30.5879974,Y 660.460266,Z 1.50000,A 0.0,B 0.0,C -20.0000},Welding_Power 58.0000,Welding_Speed 0.0200000,Welding_Angle -20.0000,Welding_CDIS 5,Welding_ACC 100,Welding_Offset {X 0.0,Y 0.0,Z -1.00000}}
C225_Welding_Craft[2,1]={Welding_Name[] "C225_S1",Welding_Pos {X 18.8446884,Y 648.925,Z 1.50000,A 0.0,B -20.0000,C 0.0},Welding_Power 60.0000,Welding_Speed 0.0430000,Welding_Angle -20.0000,Welding_CDIS 5,Welding_ACC 100,Welding_Offset {X -0.200000,Y 0.0,Z 0.0}}
C225_Welding_Craft[2,2]={Welding_Name[] "PM5",Welding_Pos {X 22.5580,Y 657.093,Z 1.50000,A 0.0,B 0.0,C 0.0},Welding_Power 60.0000,Welding_Speed 0.0400000,Welding_Angle -20.0000,Welding_CDIS 5,Welding_ACC 100,Welding_Offset {X 0.0,Y 0.700000,Z 0.0},Welding_Offset_CIR {C_X 0.0,C_Y 0.0,C_Z 0.0}}
C225_Welding_Craft[2,3]={Welding_Name[] "PE5",Welding_Pos {X 30.8369904,Y 660.939636,Z 1.50000,A 0.0,B 0.0,C -20.0000},Welding_Power 60.0000,Welding_Speed 0.0200000,Welding_Angle -20.0000,Welding_CDIS 5,Welding_ACC 100,Welding_Offset {X 0.0,Y 0.0,Z -1.00000}}

DECL GLOBAL Surr_Welding_Craft_Type L270_Welding_Craft[2,10]
L270_Welding_Craft[1,1]={Welding_Name[] "L270_S1",Welding_Pos {X 63.8416977,Y 660.477722,Z 1.50000,A 0.0,B 0.0,C -20.0000},Welding_Power 58.0000,Welding_Speed 0.0400000,Welding_Angle -20.0000,Welding_CDIS 5,Welding_ACC 100,Welding_Offset {X 0.0,Y 0.0,Z 0.0}}
L270_Welding_Craft[1,2]={Welding_Name[] "L270_S2",Welding_Pos {X 196.856491,Y 660.547485,Z 1.50000,A 0.0,B 0.0,C -20.0000},Welding_Power 58.0000,Welding_Speed 0.0400000,Welding_Angle -20.0000,Welding_CDIS 5,Welding_ACC 100,Welding_Offset {X 0.0,Y -0.300000,Z 0.0}}
L270_Welding_Craft[1,3]={Welding_Name[] "L270_S3",Welding_Pos {X 346.498108,Y 660.626,Z 1.50000,A 0.0,B 0.0,C -20.0000},Welding_Power 58.0000,Welding_Speed 0.0400000,Welding_Angle -20.0000,Welding_CDIS 5,Welding_ACC 100,Welding_Offset {X 0.0,Y -0.500000,Z 0.0}}
L270_Welding_Craft[1,4]={Welding_Name[] "S4",Welding_Pos {X 400.000,Y 86.0000153,Z -3.00000,A 0.0,B 23.0000,C 0.0},Welding_Power 80.0000,Welding_Speed 0.0400000,Welding_Angle -20.0000,Welding_CDIS 5,Welding_ACC 100,Welding_Offset {X 0.0,Y 0.0,Z 0.0}}
L270_Welding_Craft[1,5]={Welding_Name[] "S12",Welding_Pos {X 28.9999981,Y 400.000,Z -3.00000,A 0.0,B 0.0,C -23.0000},Welding_Power 80.0000,Welding_Speed 0.0400000,Welding_Angle -20.0000,Welding_CDIS 5,Welding_ACC 100,Welding_Offset {X 0.0,Y 0.0,Z 0.0}}
L270_Welding_Craft[1,6]={Welding_Name[] "S6",Welding_Pos {X 533.000,Y 463.600037,Z -2.05000,A 0.0,B -23.0000,C 0.0},Welding_Power 80.0000,Welding_Speed 0.0400000,Welding_Angle -20.0000,Welding_CDIS 5,Welding_ACC 100,Welding_Offset {X 0.0,Y 0.0,Z 0.0}}
L270_Welding_Craft[1,7]={Welding_Name[] "S7",Welding_Pos {X 533.000,Y 463.600037,Z -2.05000,A 0.0,B -23.0000,C 0.0},Welding_Power 80.0000,Welding_Speed 0.0400000,Welding_Angle -20.0000,Welding_CDIS 5,Welding_ACC 100,Welding_Offset {X 0.0,Y 0.0,Z 0.0}}
L270_Welding_Craft[1,8]={Welding_Name[] "S8",Welding_Pos {X 533.000,Y 463.600037,Z -2.05000,A 0.0,B -23.0000,C 0.0},Welding_Power 80.0000,Welding_Speed 0.0400000,Welding_Angle -20.0000,Welding_CDIS 5,Welding_ACC 100,Welding_Offset {X 0.0,Y 0.0,Z 0.0}}
L270_Welding_Craft[1,9]={Welding_Name[] "S9",Welding_Pos {X 533.000,Y 463.600037,Z -2.05000,A 0.0,B -23.0000,C 0.0},Welding_Power 80.0000,Welding_Speed 0.0400000,Welding_Angle -20.0000,Welding_CDIS 5,Welding_ACC 100,Welding_Offset {X 0.0,Y 0.0,Z 0.0}}
L270_Welding_Craft[1,10]={Welding_Name[] "S10",Welding_Pos {X 533.000,Y 338.000,Z -2.05000,A 0.0,B -23.0000,C 0.0},Welding_Power 80.0000,Welding_Speed 0.0400000,Welding_Angle -20.0000,Welding_CDIS 5,Welding_ACC 100,Welding_Offset {X 0.0,Y 0.0,Z 0.0}}
L270_Welding_Craft[2,1]={Welding_Name[] "L270_S1",Welding_Pos {X 64.1063919,Y 660.980286,Z 1.50000,A 0.0,B 0.0,C -20.0000},Welding_Power 60.0000,Welding_Speed 0.0450000,Welding_Angle -20.0000,Welding_CDIS 5,Welding_ACC 100,Welding_Offset {X 0.0,Y -0.100000,Z -1.00000}}
L270_Welding_Craft[2,2]={Welding_Name[] "L270_S2",Welding_Pos {X 197.184,Y 661.143,Z 1.50000,A 0.0,B 0.0,C -20.0000},Welding_Power 60.0000,Welding_Speed 0.0450000,Welding_Angle -20.0000,Welding_CDIS 5,Welding_ACC 100,Welding_Offset {X 0.0,Y -0.300000,Z 0.0}}
L270_Welding_Craft[2,3]={Welding_Name[] "L270_S3",Welding_Pos {X 346.896301,Y 661.326050,Z 1.50000,A 0.0,B 0.0,C -20.0000},Welding_Power 60.0000,Welding_Speed 0.0450000,Welding_Angle -20.0000,Welding_CDIS 5,Welding_ACC 100,Welding_Offset {X 0.0,Y -0.400000,Z 0.0}}
L270_Welding_Craft[2,4]={Welding_Name[] "S4",Welding_Pos {X 400.000,Y 86.0000153,Z -3.00000,A 0.0,B 23.0000,C 0.0},Welding_Power 80.0000,Welding_Speed 0.0400000,Welding_Angle -20.0000,Welding_CDIS 5,Welding_ACC 100,Welding_Offset {X 0.0,Y 0.0,Z 0.0}}
L270_Welding_Craft[2,5]={Welding_Name[] "S12",Welding_Pos {X 28.9999981,Y 400.000,Z -3.00000,A 0.0,B 0.0,C -23.0000},Welding_Power 80.0000,Welding_Speed 0.0400000,Welding_Angle -20.0000,Welding_CDIS 5,Welding_ACC 100,Welding_Offset {X 0.0,Y 0.0,Z 0.0}}
L270_Welding_Craft[2,6]={Welding_Name[] "S6",Welding_Pos {X 533.000,Y 463.600037,Z -2.05000,A 0.0,B -23.0000,C 0.0},Welding_Power 80.0000,Welding_Speed 0.0400000,Welding_Angle -20.0000,Welding_CDIS 5,Welding_ACC 100,Welding_Offset {X 0.0,Y 0.0,Z 0.0}}
L270_Welding_Craft[2,7]={Welding_Name[] "S7",Welding_Pos {X 533.000,Y 463.600037,Z -2.05000,A 0.0,B -23.0000,C 0.0},Welding_Power 80.0000,Welding_Speed 0.0400000,Welding_Angle -20.0000,Welding_CDIS 5,Welding_ACC 100,Welding_Offset {X 0.0,Y 0.0,Z 0.0}}
L270_Welding_Craft[2,8]={Welding_Name[] "S8",Welding_Pos {X 533.000,Y 463.600037,Z -2.05000,A 0.0,B -23.0000,C 0.0},Welding_Power 80.0000,Welding_Speed 0.0400000,Welding_Angle -20.0000,Welding_CDIS 5,Welding_ACC 100,Welding_Offset {X 0.0,Y 0.0,Z 0.0}}
L270_Welding_Craft[2,9]={Welding_Name[] "S9",Welding_Pos {X 533.000,Y 463.600037,Z -2.05000,A 0.0,B -23.0000,C 0.0},Welding_Power 80.0000,Welding_Speed 0.0400000,Welding_Angle -20.0000,Welding_CDIS 5,Welding_ACC 100,Welding_Offset {X 0.0,Y 0.0,Z 0.0}}
L270_Welding_Craft[2,10]={Welding_Name[] "S10",Welding_Pos {X 533.000,Y 338.000,Z -2.05000,A 0.0,B -23.0000,C 0.0},Welding_Power 80.0000,Welding_Speed 0.0400000,Welding_Angle -20.0000,Welding_CDIS 5,Welding_ACC 100,Welding_Offset {X 0.0,Y 0.0,Z 0.0}}

DECL GLOBAL Surr_Welding_Craft_Type C315_Welding_Craft[2,3]
C315_Welding_Craft[1,1]={Welding_Name[] "C315_S1",Welding_Pos {X 363.125,Y 660.634705,Z 1.50000,A 0.0,B 0.0,C -20.0000},Welding_Power 80.0000,Welding_Speed 0.0400000,Welding_Angle -20.0000,Welding_CDIS 5,Welding_ACC 100,Welding_Offset {X 0.0,Y -0.700000,Z -1.00000}}
C315_Welding_Craft[1,2]={Welding_Name[] "PM7",Welding_Pos {X 370.778,Y 657.395,Z 1.50000,A 0.0,B 0.0,C 0.0},Welding_Power 80.0000,Welding_Speed 0.0400000,Welding_Angle 20.0000,Welding_CDIS 5,Welding_ACC 100,Welding_Offset {X 0.0,Y 0.0,Z -1.00000},Welding_Offset_CIR {C_X 0.0,C_Y 0.0,C_Z 0.0}}
C315_Welding_Craft[1,3]={Welding_Name[] "PE7",Welding_Pos {X 375.130585,Y 648.641,Z 1.50000,A 0.0,B 20.0000,C 0.0},Welding_Power 58.0000,Welding_Speed 0.0200000,Welding_Angle 20.0000,Welding_CDIS 5,Welding_ACC 100,Welding_Offset {X -1.00000,Y -0.700000,Z -1.00000}}
C315_Welding_Craft[2,1]={Welding_Name[] "C315_S1",Welding_Pos {X 363.531,Y 661.346375,Z 1.50000,A 0.0,B 0.0,C -20.0000},Welding_Power 60.0000,Welding_Speed 0.0300000,Welding_Angle -20.0000,Welding_CDIS -1,Welding_ACC 80,Welding_Offset {X 0.0,Y -0.500000,Z -1.50000}}
C315_Welding_Craft[2,2]={Welding_Name[] "PM7",Welding_Pos {X 371.252,Y 658.128,Z 1.50000,A 0.0,B 0.0,C 0.0},Welding_Power 54.0000,Welding_Speed 0.0400000,Welding_Angle 20.0000,Welding_CDIS 5,Welding_ACC 100,Welding_Offset {X -0.300000,Y 0.0,Z 1.00000},Welding_Offset_CIR {C_X 0.0,C_Y 0.0,C_Z 0.0}}
C315_Welding_Craft[2,3]={Welding_Name[] "PE7",Welding_Pos {X 375.537689,Y 649.361,Z 1.50000,A 0.0,B 20.0000,C 0.0},Welding_Power 54.0000,Welding_Speed 0.0200000,Welding_Angle 20.0000,Welding_CDIS 5,Welding_ACC 100,Welding_Offset {X -0.100000,Y -0.100000,Z 1.00000}}


DECL GLOBAL Surr_Welding_Craft_Type N45_Short_Craft[2,5]
N45_Short_Craft[1,1]={Welding_Name[] "S5",Welding_Pos {X 364.000,Y 0.0,Z -150.000,A 0.0,B 0.0,C 0.0},Welding_Power 80.0000,Welding_Speed 0.500000,Welding_Angle 0.0,Welding_CDIS 0,Welding_ACC 100,Welding_Offset {X 0.0,Y 0.0,Z 0.0}}
N45_Short_Craft[1,2]={Welding_Name[] "S13",Welding_Pos {X 364.000,Y 0.0,Z 0.0,A 0.0,B 0.0,C 0.0},Welding_Power 80.0000,Welding_Speed 0.500000,Welding_Angle 0.0,Welding_CDIS 0,Welding_ACC 100,Welding_Offset {X 0.0,Y 0.0,Z 0.0}}
N45_Short_Craft[1,3]={Welding_Name[] "S14",Welding_Pos {X 364.000,Y 23.0000,Z 0.0,A 0.0,B 0.0,C 0.0},Welding_Power 80.0000,Welding_Speed 0.01000000,Welding_Angle 0.0,Welding_CDIS 0,Welding_ACC 100,Welding_Offset {X 0.0,Y 0.0,Z 0.0}}
N45_Short_Craft[1,4]={Welding_Name[] "S4",Welding_Pos {X 364.000,Y 20.7000,Z -150.000,A 0.0,B 0.0,C 0.0},Welding_Power 80.0000,Welding_Speed 0.500000,Welding_Angle 0.0,Welding_CDIS 0,Welding_ACC 100,Welding_Offset {X 0.0,Y 0.0,Z 0.0}}
N45_Short_Craft[1,5]={Welding_Name[] "S12",Welding_Pos {X 28.9999981,Y 400.000,Z -3.00000,A 0.0,B 0.0,C -23.0000},Welding_Power 80.0000,Welding_Speed 0.500000,Welding_Angle 0.0,Welding_CDIS 0,Welding_ACC 100,Welding_Offset {X 0.0,Y 0.0,Z 0.0}}
N45_Short_Craft[2,1]={Welding_Name[] "S5",Welding_Pos {X 362.596,Y -0.482000,Z -150.000,A 0.0,B 0.0,C 0.0},Welding_Power 80.0000,Welding_Speed 0.500000,Welding_Angle 0.0,Welding_CDIS 0,Welding_ACC 100,Welding_Offset {X 0.0,Y 0.0,Z 0.0}}
N45_Short_Craft[2,2]={Welding_Name[] "S13",Welding_Pos {X 362.596,Y -0.482000,Z 0.0,A 0.0,B 0.0,C 0.0},Welding_Power 80.0000,Welding_Speed 0.500000,Welding_Angle 0.0,Welding_CDIS 0,Welding_ACC 100,Welding_Offset {X 0.0,Y 0.0,Z 0.0}}
N45_Short_Craft[2,3]={Welding_Name[] "S14",Welding_Pos {X 362.546,Y 18.7470,Z 0.0,A 0.0,B 0.0,C 0.0},Welding_Power 80.0000,Welding_Speed 0.01000000,Welding_Angle 0.0,Welding_CDIS 0,Welding_ACC 100,Welding_Offset {X 0.0,Y 0.0,Z 0.0}}
N45_Short_Craft[2,4]={Welding_Name[] "S4",Welding_Pos {X 362.566040,Y 11.0408678,Z -150.000,A 0.0,B 0.0,C 0.0},Welding_Power 80.0000,Welding_Speed 0.500000,Welding_Angle 0.0,Welding_CDIS 0,Welding_ACC 100,Welding_Offset {X 0.0,Y 0.0,Z 0.0}}
N45_Short_Craft[2,5]={Welding_Name[] "S12",Welding_Pos {X 28.9999981,Y 400.000,Z -3.00000,A 0.0,B 0.0,C -23.0000},Welding_Power 80.0000,Welding_Speed 0.500000,Welding_Angle 0.0,Welding_CDIS 0,Welding_ACC 100,Welding_Offset {X 0.0,Y 0.0,Z 0.0}}

DECL GLOBAL Surr_Welding_Craft_Type N135_Short_Craft[2,5]
N135_Short_Craft[1,1]={Welding_Name[] "S9",Welding_Pos {X 36.0000,Y 0.0,Z -150.000,A 0.0,B 0.0,C 0.0},Welding_Power 80.0000,Welding_Speed 0.500000,Welding_Angle 0.0,Welding_CDIS 0,Welding_ACC 100,Welding_Offset {X 0.0,Y 0.0,Z 0.0}}
N135_Short_Craft[1,2]={Welding_Name[] "S13",Welding_Pos {X 36.0000,Y 0.0,Z 0.0,A 0.0,B 0.0,C 0.0},Welding_Power 80.0000,Welding_Speed 0.500000,Welding_Angle 0.0,Welding_CDIS 0,Welding_ACC 100,Welding_Offset {X 0.0,Y 0.0,Z 0.0}}
N135_Short_Craft[1,3]={Welding_Name[] "S14",Welding_Pos {X 36.0000,Y 23.0000,Z 0.0,A 0.0,B 0.0,C 0.0},Welding_Power 80.0000,Welding_Speed 0.01000000,Welding_Angle 0.0,Welding_CDIS 0,Welding_ACC 100,Welding_Offset {X 0.0,Y 0.0,Z 0.0}}
N135_Short_Craft[1,4]={Welding_Name[] "S4",Welding_Pos {X 36.0000,Y 20.7000,Z -150.000,A 0.0,B 0.0,C 0.0},Welding_Power 80.0000,Welding_Speed 0.500000,Welding_Angle 0.0,Welding_CDIS 0,Welding_ACC 100,Welding_Offset {X 0.0,Y 0.0,Z 0.0}}
N135_Short_Craft[1,5]={Welding_Name[] "S12",Welding_Pos {X 28.9999981,Y 400.000,Z -3.00000,A 0.0,B 0.0,C -23.0000},Welding_Power 80.0000,Welding_Speed 0.500000,Welding_Angle 0.0,Welding_CDIS 0,Welding_ACC 100,Welding_Offset {X 0.0,Y 0.0,Z 0.0}}
N135_Short_Craft[2,1]={Welding_Name[] "S9",Welding_Pos {X 32.1370,Y -0.736000,Z -150.000,A 0.0,B 0.0,C 0.0},Welding_Power 80.0000,Welding_Speed 0.500000,Welding_Angle 0.0,Welding_CDIS 0,Welding_ACC 100,Welding_Offset {X 0.0,Y 0.0,Z 0.0}}
N135_Short_Craft[2,2]={Welding_Name[] "S13",Welding_Pos {X 32.1370,Y -0.736000,Z 0.0,A 0.0,B 0.0,C 0.0},Welding_Power 80.0000,Welding_Speed 0.500000,Welding_Angle 0.0,Welding_CDIS 0,Welding_ACC 100,Welding_Offset {X 0.0,Y 0.0,Z 0.0}}
N135_Short_Craft[2,3]={Welding_Name[] "S14",Welding_Pos {X 32.1600,Y 18.4470,Z 0.0,A 0.0,B 0.0,C 0.0},Welding_Power 80.0000,Welding_Speed 0.01000000,Welding_Angle 0.0,Welding_CDIS 0,Welding_ACC 100,Welding_Offset {X 0.0,Y 0.0,Z 0.0}}
N135_Short_Craft[2,4]={Welding_Name[] "S4",Welding_Pos {X 32.1485,Y 8.85550117,Z -150.000,A 0.0,B 0.0,C 0.0},Welding_Power 80.0000,Welding_Speed 0.500000,Welding_Angle 0.0,Welding_CDIS 0,Welding_ACC 100,Welding_Offset {X 0.0,Y 0.0,Z 0.0}}
N135_Short_Craft[2,5]={Welding_Name[] "S12",Welding_Pos {X 28.9999981,Y 400.000,Z -3.00000,A 0.0,B 0.0,C -23.0000},Welding_Power 80.0000,Welding_Speed 0.500000,Welding_Angle 0.0,Welding_CDIS 0,Welding_ACC 100,Welding_Offset {X 0.0,Y 0.0,Z 0.0}}

DECL GLOBAL Surr_Welding_Craft_Type N225_Short_Craft[2,5]
N225_Short_Craft[1,1]={Welding_Name[] "S13",Welding_Pos {X 36.0000,Y 680.000,Z -150.000,A 0.0,B 0.0,C 0.0},Welding_Power 80.0000,Welding_Speed 0.500000,Welding_Angle 0.0,Welding_CDIS 0,Welding_ACC 100,Welding_Offset {X 0.0,Y 0.0,Z 0.0}}
N225_Short_Craft[1,2]={Welding_Name[] "S13",Welding_Pos {X 36.0000,Y 680.000,Z 0.0,A 0.0,B 0.0,C 0.0},Welding_Power 80.0000,Welding_Speed 0.500000,Welding_Angle 0.0,Welding_CDIS 0,Welding_ACC 100,Welding_Offset {X 0.0,Y 0.0,Z 0.0}}
N225_Short_Craft[1,3]={Welding_Name[] "S14",Welding_Pos {X 36.0000,Y 657.000,Z 0.0,A 0.0,B 0.0,C 0.0},Welding_Power 80.0000,Welding_Speed 0.01000000,Welding_Angle 0.0,Welding_CDIS 0,Welding_ACC 100,Welding_Offset {X 0.0,Y 0.0,Z 0.0}}
N225_Short_Craft[1,4]={Welding_Name[] "S4",Welding_Pos {X 36.0000,Y 667.500,Z -150.000,A 0.0,B 0.0,C 0.0},Welding_Power 80.0000,Welding_Speed 0.500000,Welding_Angle 0.0,Welding_CDIS 0,Welding_ACC 100,Welding_Offset {X 0.0,Y 0.0,Z 0.0}}
N225_Short_Craft[1,5]={Welding_Name[] "S12",Welding_Pos {X 28.9999981,Y 400.000,Z -3.00000,A 0.0,B 0.0,C -23.0000},Welding_Power 80.0000,Welding_Speed 0.500000,Welding_Angle 0.0,Welding_CDIS 0,Welding_ACC 100,Welding_Offset {X 0.0,Y 0.0,Z 0.0}}
N225_Short_Craft[2,1]={Welding_Name[] "S13",Welding_Pos {X 31.6630,Y 678.803,Z -150.000,A 0.0,B 0.0,C 0.0},Welding_Power 80.0000,Welding_Speed 0.500000,Welding_Angle 0.0,Welding_CDIS 0,Welding_ACC 100,Welding_Offset {X 0.0,Y 0.0,Z 0.0}}
N225_Short_Craft[2,2]={Welding_Name[] "S13",Welding_Pos {X 31.6630,Y 678.803,Z 0.0,A 0.0,B 0.0,C 0.0},Welding_Power 80.0000,Welding_Speed 0.500000,Welding_Angle 0.0,Welding_CDIS 0,Welding_ACC 100,Welding_Offset {X 0.0,Y 0.0,Z 0.0}}
N225_Short_Craft[2,3]={Welding_Name[] "S14",Welding_Pos {X 31.3610,Y 659.596,Z 0.0,A 0.0,B 0.0,C 0.0},Welding_Power 80.0000,Welding_Speed 0.01000000,Welding_Angle 0.0,Welding_CDIS 0,Welding_ACC 100,Welding_Offset {X 0.0,Y 0.0,Z 0.0}}
N225_Short_Craft[2,4]={Welding_Name[] "S4",Welding_Pos {X 31.5120010,Y 669.199463,Z -150.000,A 0.0,B 0.0,C 0.0},Welding_Power 80.0000,Welding_Speed 0.500000,Welding_Angle 0.0,Welding_CDIS 0,Welding_ACC 100,Welding_Offset {X 0.0,Y 0.0,Z 0.0}}
N225_Short_Craft[2,5]={Welding_Name[] "S12",Welding_Pos {X 28.9999981,Y 400.000,Z -3.00000,A 0.0,B 0.0,C -23.0000},Welding_Power 80.0000,Welding_Speed 0.500000,Welding_Angle 0.0,Welding_CDIS 0,Welding_ACC 100,Welding_Offset {X 0.0,Y 0.0,Z 0.0}}

DECL GLOBAL Surr_Welding_Craft_Type N315_Short_Craft[2,5]
N315_Short_Craft[1,1]={Welding_Name[] "S17",Welding_Pos {X 364.000,Y 680.000,Z -150.000,A 0.0,B 0.0,C 0.0},Welding_Power 80.0000,Welding_Speed 0.500000,Welding_Angle 0.0,Welding_CDIS 0,Welding_ACC 100,Welding_Offset {X 0.0,Y 0.0,Z 0.0}}
N315_Short_Craft[1,2]={Welding_Name[] "S13",Welding_Pos {X 364.000,Y 680.000,Z 0.0,A 0.0,B 0.0,C 0.0},Welding_Power 80.0000,Welding_Speed 0.500000,Welding_Angle 0.0,Welding_CDIS 0,Welding_ACC 100,Welding_Offset {X 0.0,Y 0.0,Z 0.0}}
N315_Short_Craft[1,3]={Welding_Name[] "S14",Welding_Pos {X 364.000,Y 657.000,Z 0.0,A 0.0,B 0.0,C 0.0},Welding_Power 80.0000,Welding_Speed 0.01000000,Welding_Angle 0.0,Welding_CDIS 0,Welding_ACC 100,Welding_Offset {X 0.0,Y 0.0,Z 0.0}}
N315_Short_Craft[1,4]={Welding_Name[] "S4",Welding_Pos {X 364.000,Y 667.500,Z -150.000,A 0.0,B 0.0,C 0.0},Welding_Power 80.0000,Welding_Speed 0.500000,Welding_Angle 0.0,Welding_CDIS 0,Welding_ACC 100,Welding_Offset {X 0.0,Y 0.0,Z 0.0}}
N315_Short_Craft[1,5]={Welding_Name[] "S12",Welding_Pos {X 28.9999981,Y 400.000,Z -3.00000,A 0.0,B 0.0,C -23.0000},Welding_Power 80.0000,Welding_Speed 0.500000,Welding_Angle 0.0,Welding_CDIS 0,Welding_ACC 100,Welding_Offset {X 0.0,Y 0.0,Z 0.0}}
N315_Short_Craft[2,1]={Welding_Name[] "S17",Welding_Pos {X 361.885,Y 679.437,Z -150.000,A 0.0,B 0.0,C 0.0},Welding_Power 80.0000,Welding_Speed 0.500000,Welding_Angle 0.0,Welding_CDIS 0,Welding_ACC 100,Welding_Offset {X 0.0,Y 0.0,Z 0.0}}
N315_Short_Craft[2,2]={Welding_Name[] "S13",Welding_Pos {X 361.885,Y 679.437,Z 0.0,A 0.0,B 0.0,C 0.0},Welding_Power 80.0000,Welding_Speed 0.500000,Welding_Angle 0.0,Welding_CDIS 0,Welding_ACC 100,Welding_Offset {X 0.0,Y 0.0,Z 0.0}}
N315_Short_Craft[2,3]={Welding_Name[] "S14",Welding_Pos {X 361.560,Y 660.457,Z 0.0,A 0.0,B 0.0,C 0.0},Welding_Power 80.0000,Welding_Speed 0.01000000,Welding_Angle 0.0,Welding_CDIS 0,Welding_ACC 100,Welding_Offset {X 0.0,Y 0.0,Z 0.0}}
N315_Short_Craft[2,4]={Welding_Name[] "S4",Welding_Pos {X 361.722504,Y 669.947,Z -150.000,A 0.0,B 0.0,C 0.0},Welding_Power 80.0000,Welding_Speed 0.500000,Welding_Angle 0.0,Welding_CDIS 0,Welding_ACC 100,Welding_Offset {X 0.0,Y 0.0,Z 0.0}}
N315_Short_Craft[2,5]={Welding_Name[] "S12",Welding_Pos {X 28.9999981,Y 400.000,Z -3.00000,A 0.0,B 0.0,C -23.0000},Welding_Power 80.0000,Welding_Speed 0.500000,Welding_Angle 0.0,Welding_CDIS 0,Welding_ACC 100,Welding_Offset {X 0.0,Y 0.0,Z 0.0}}

DECL GLOBAL E6POS Vision_Result_POS={X 175.013321,Y -792.138306,Z 222.764145,A 0.0,B 0.0,C 0.0}


DECL GLOBAL Surround_Welding_Type N1_Sink_Data={Sink_Size_Long 640.000,Sink_Size_Width 355.000,Sink_Size_R 12.0000,Sink_Size_Short_Side 20.0000,Sink_Size_Short_OnePos 31.2000,Sink_Size_Short_TwoPos 332.700,Sink_Size_Pots_Thick 0.0,Sink_Size_Panel_Thick -1.50000,Sink_Model 902182,Sink_Size_Left_Distance 20.0000,Sink_Size_Down_Distance 20.0000,Sink_Type #LeftRight_One}
DECL GLOBAL Surround_Welding_Type N2_Sink_Data={Sink_Size_Long 640.000,Sink_Size_Width 355.000,Sink_Size_R 12.0000,Sink_Size_Short_Side 20.0000,Sink_Size_Short_OnePos 31.2000,Sink_Size_Short_TwoPos 332.700,Sink_Size_Pots_Thick 0.0,Sink_Size_Panel_Thick -1.50000,Sink_Model 902182,Sink_Size_Left_Distance 20.0000,Sink_Size_Down_Distance 20.0000,Sink_Type #LeftRight_One}
;-----------Viion_INI------------



DECL GLOBAL INT Vision_Scope=20
DECL GLOBAL REAL Vision_Trans_Max_Offset=20.0000
DECL GLOBAL REAL Vision_Rota_Max_Offset=5.00000
DECL GLOBAL Vision_Type_Enum Vision_Type=#Vision_Text
;GLOBAL CHAR $Socket_Connect[1024]
;DECL GLOBAL CHAR $SOCKET_MESS[1024]
;DECL GLOBAL MODEL_TYPE $N_1
;DECL GLOBAL MODEL_TYPE $N_2
;DECL GLOBAL INT $MY_Work_Number=-1
DECL GLOBAL BOOL Vision_OFFSET_STATE=TRUE


;----------------------------------
ENDDAT
